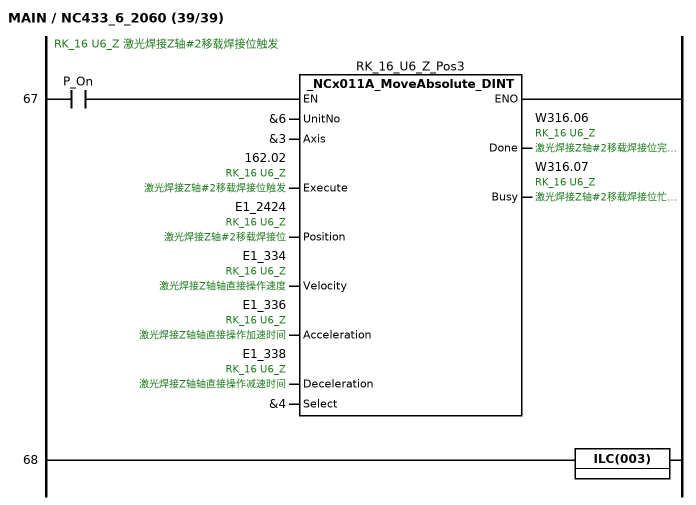
; [picture p264: MAIN / NC433_6_2060, rungs 67-68]
; rung 67: RK_16 U6_Z 激光焊接Z轴#2移载焊接位触发
LD P_On
CALL RK_16_U6_Z_Pos3 : _NCx011A_MoveAbsolute_DINT (UnitNo := &6, Axis := &3, Execute := 162.02, Position := E1_2424, Velocity := E1_334, Acceleration := E1_336, Deceleration := E1_338, Select := &4, Done => W316.06, Busy => W316.07)  ; RK_16 U6_Z 激光焊接Z轴#2移载焊接位触发, RK_16 U6_Z 激光焊接Z轴#2移载焊接位, RK_16 U6_Z 激光焊接Z轴轴直接操作速度, RK_16 U6_Z 激光焊接Z轴轴直接操作加速时间, RK_16 U6_Z 激光焊接Z轴轴直接操作减速时间, RK_16 U6_Z 激光焊接Z轴#2移载焊接位完成标志, RK_16 U6_Z 激光焊接Z轴#2移载焊接位忙标志
; rung 68
ILC(003)

### Section NC433_8_2080

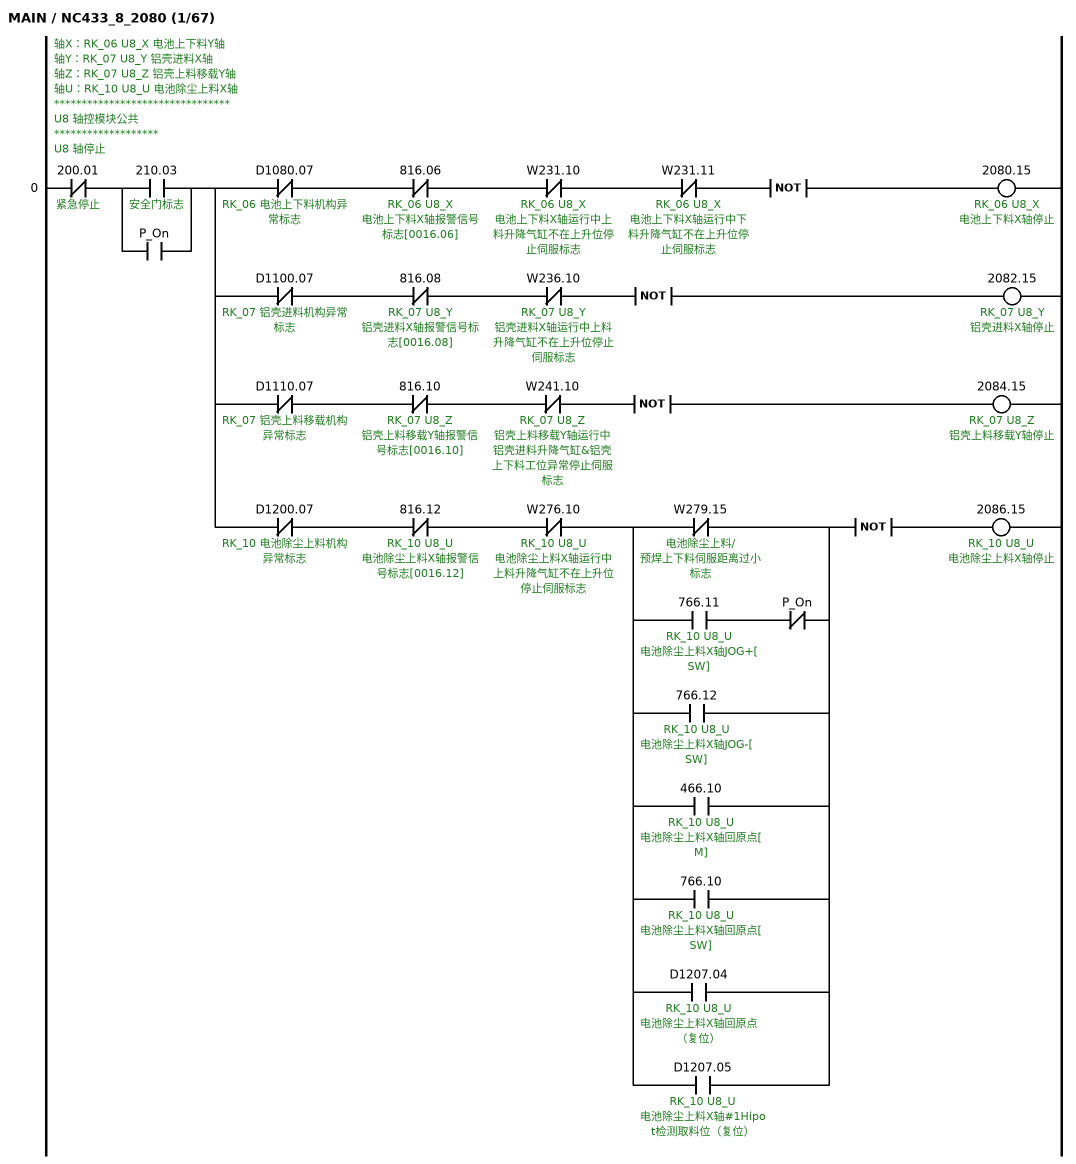
; rung 0: 轴X：RK_06 U8_X 电池上下料Y轴 / 轴Y：RK_07 U8_Y 铝壳进料X轴 / 轴Z：RK_07 U8_Z 铝壳上料移载Y轴 / 轴U：RK_10 U8_U 电池除尘上料X轴 / ******************************** / U8 轴控模块公共 / ******************* / U8 轴停止
LDNOT 200.01  ; 紧急停止
LD 210.03  ; 安全门标志
OR P_On
ANDLD
OUT TR0
ANDNOT D1080.07  ; RK_06 电池上下料机构异常标志
ANDNOT 816.06  ; RK_06 U8_X 电池上下料X轴报警信号标志[0016.06]
ANDNOT W231.10  ; RK_06 U8_X 电池上下料X轴运行中上料升降气缸不在上升位停止伺服标志
ANDNOT W231.11  ; RK_06 U8_X 电池上下料X轴运行中下料升降气缸不在上升位停止伺服标志
NOT(520)
OUT 2080.15  ; RK_06 U8_X 电池上下料X轴停止
LD TR0
ANDNOT D1100.07  ; RK_07 铝壳进料机构异常标志
ANDNOT 816.08  ; RK_07 U8_Y 铝壳进料X轴报警信号标志[0016.08]
ANDNOT W236.10  ; RK_07 U8_Y 铝壳进料X轴运行中上料升降气缸不在上升位停止伺服标志
NOT(520)
OUT 2082.15  ; RK_07 U8_Y 铝壳进料X轴停止
LD TR0
ANDNOT D1110.07  ; RK_07 铝壳上料移载机构异常标志
ANDNOT 816.10  ; RK_07 U8_Z 铝壳上料移载Y轴报警信号标志[0016.10]
ANDNOT W241.10  ; RK_07 U8_Z 铝壳上料移载Y轴运行中铝壳进料升降气缸&铝壳上下料工位异常停止伺服标志
NOT(520)
OUT 2084.15  ; RK_07 U8_Z 铝壳上料移载Y轴停止
LD TR0
ANDNOT D1200.07  ; RK_10 电池除尘上料机构异常标志
ANDNOT 816.12  ; RK_10 U8_U 电池除尘上料X轴报警信号标志[0016.12]
ANDNOT W276.10  ; RK_10 U8_U 电池除尘上料X轴运行中上料升降气缸不在上升位停止伺服标志
LDNOT W279.15  ; 电池除尘上料/预焊上下料伺服距离过小标志
LD 766.11  ; RK_10 U8_U 电池除尘上料X轴JOG+[SW]
ANDNOT P_On
ORLD
OR 766.12  ; RK_10 U8_U 电池除尘上料X轴JOG-[SW]
OR 466.10  ; RK_10 U8_U 电池除尘上料X轴回原点[M]
OR 766.10  ; RK_10 U8_U 电池除尘上料X轴回原点[SW]
OR D1207.04  ; RK_10 U8_U 电池除尘上料X轴回原点（复位）
OR D1207.05  ; RK_10 U8_U 电池除尘上料X轴#1Hipot检测取料位（复位）
ANDLD
NOT(520)
OUT 2086.15  ; RK_10 U8_U 电池除尘上料X轴停止

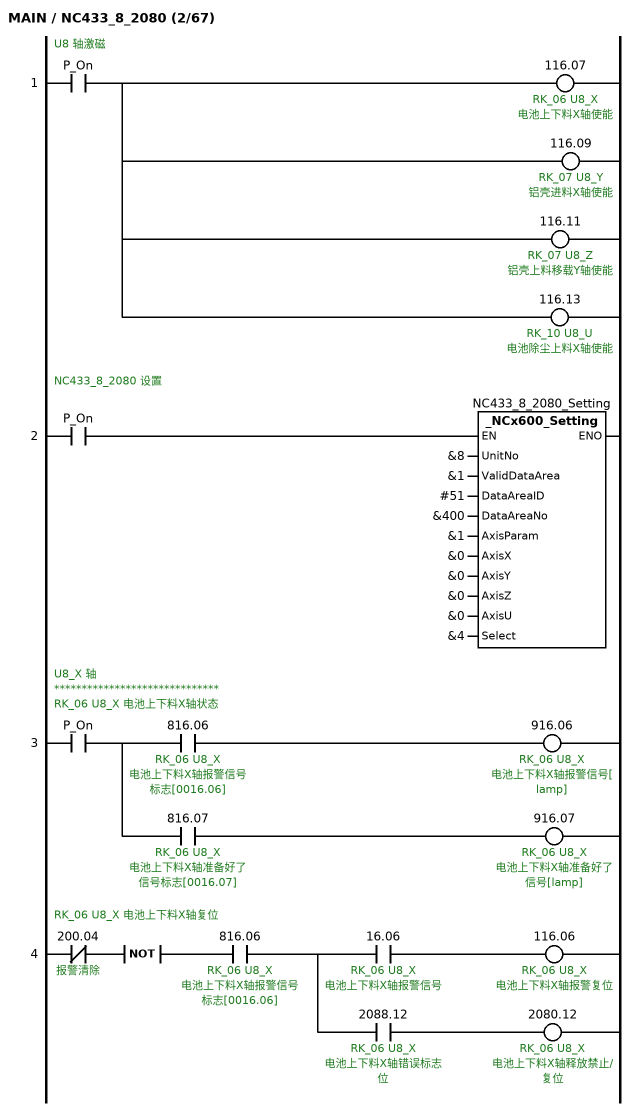
; rung 1: U8 轴激磁
LD P_On
OUT 116.07  ; RK_06 U8_X 电池上下料X轴使能
OUT 116.09  ; RK_07 U8_Y 铝壳进料X轴使能
OUT 116.11  ; RK_07 U8_Z 铝壳上料移载Y轴使能
OUT 116.13  ; RK_10 U8_U 电池除尘上料X轴使能
; rung 2: NC433_8_2080 设置
LD P_On
CALL NC433_8_2080_Setting : _NCx600_Setting (UnitNo := &8, ValidDataArea := &1, DataAreaID := #51, DataAreaNo := &400, AxisParam := &1, AxisX := &0, AxisY := &0, AxisZ := &0, AxisU := &0, Select := &4)
; rung 3: U8_X 轴 / ****************************** / RK_06 U8_X 电池上下料X轴状态
LD P_On
OUT TR0
AND 816.06  ; RK_06 U8_X 电池上下料X轴报警信号标志[0016.06]
OUT 916.06  ; RK_06 U8_X 电池上下料X轴报警信号[lamp]
LD TR0
AND 816.07  ; RK_06 U8_X 电池上下料X轴准备好了信号标志[0016.07]
OUT 916.07  ; RK_06 U8_X 电池上下料X轴准备好了信号[lamp]
; rung 4: RK_06 U8_X 电池上下料X轴复位
LDNOT 200.04  ; 报警清除
NOT(520)
AND 816.06  ; RK_06 U8_X 电池上下料X轴报警信号标志[0016.06]
OUT TR0
AND 16.06  ; RK_06 U8_X 电池上下料X轴报警信号
OUT 116.06  ; RK_06 U8_X 电池上下料X轴报警复位
LD TR0
AND 2088.12  ; RK_06 U8_X 电池上下料X轴错误标志位
OUT 2080.12  ; RK_06 U8_X 电池上下料X轴释放禁止/复位

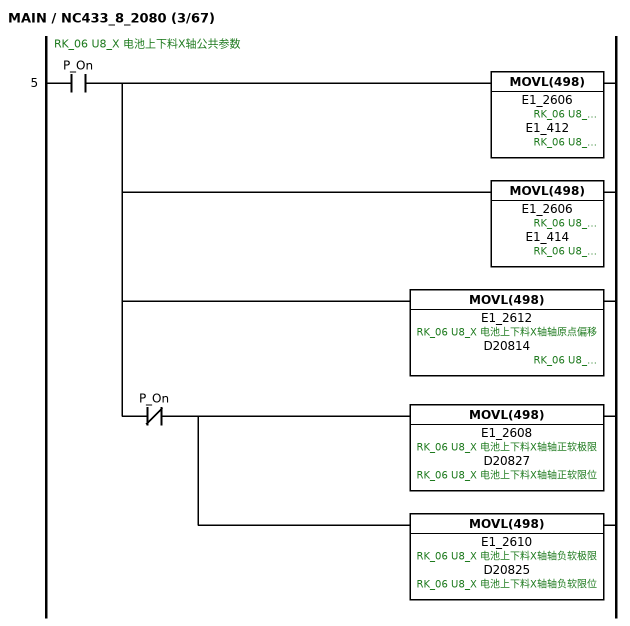
; rung 5: RK_06 U8_X 电池上下料X轴公共参数
LD P_On
MOVL(498) E1_2606 E1_412  ; RK_06 U8_X 电池上下料X轴轴加减速时间, RK_06 U8_X 电池上下料X轴轴直接操作加速时间
MOVL(498) E1_2606 E1_414  ; RK_06 U8_X 电池上下料X轴轴加减速时间, RK_06 U8_X 电池上下料X轴轴直接操作减速时间
MOVL(498) E1_2612 D20814  ; RK_06 U8_X 电池上下料X轴轴原点偏移, RK_06 U8_X 电池上下料X轴轴原点补偿值
ANDNOT P_On
MOVL(498) E1_2608 D20827  ; RK_06 U8_X 电池上下料X轴轴正软极限, RK_06 U8_X 电池上下料X轴轴正软限位
MOVL(498) E1_2610 D20825  ; RK_06 U8_X 电池上下料X轴轴负软极限, RK_06 U8_X 电池上下料X轴轴负软限位

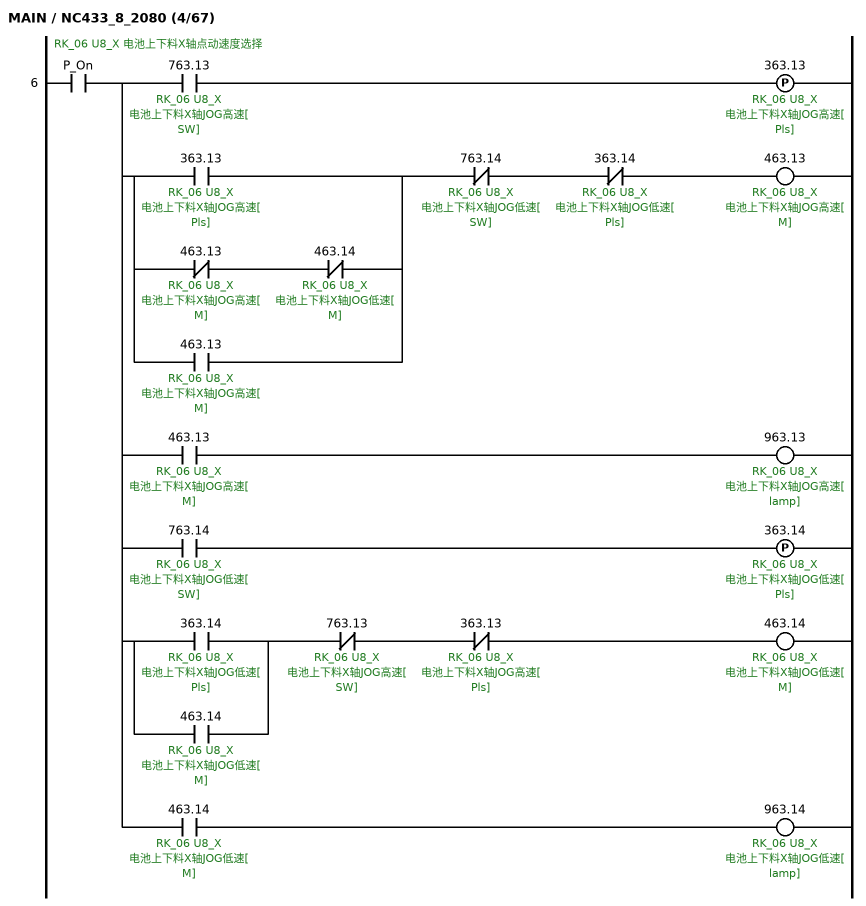
; rung 6: RK_06 U8_X 电池上下料X轴点动速度选择
LD P_On
OUT TR0
AND 763.13  ; RK_06 U8_X 电池上下料X轴JOG高速[SW]
DIFU(013) 363.13  ; RK_06 U8_X 电池上下料X轴JOG高速[Pls]
LD TR0
LD 363.13  ; RK_06 U8_X 电池上下料X轴JOG高速[Pls]
LDNOT 463.13  ; RK_06 U8_X 电池上下料X轴JOG高速[M]
ANDNOT 463.14  ; RK_06 U8_X 电池上下料X轴JOG低速[M]
ORLD
OR 463.13  ; RK_06 U8_X 电池上下料X轴JOG高速[M]
ANDLD
ANDNOT 763.14  ; RK_06 U8_X 电池上下料X轴JOG低速[SW]
ANDNOT 363.14  ; RK_06 U8_X 电池上下料X轴JOG低速[Pls]
OUT 463.13  ; RK_06 U8_X 电池上下料X轴JOG高速[M]
LD TR0
AND 463.13  ; RK_06 U8_X 电池上下料X轴JOG高速[M]
OUT 963.13  ; RK_06 U8_X 电池上下料X轴JOG高速[lamp]
LD TR0
AND 763.14  ; RK_06 U8_X 电池上下料X轴JOG低速[SW]
DIFU(013) 363.14  ; RK_06 U8_X 电池上下料X轴JOG低速[Pls]
LD TR0
LD 363.14  ; RK_06 U8_X 电池上下料X轴JOG低速[Pls]
OR 463.14  ; RK_06 U8_X 电池上下料X轴JOG低速[M]
ANDLD
ANDNOT 763.13  ; RK_06 U8_X 电池上下料X轴JOG高速[SW]
ANDNOT 363.13  ; RK_06 U8_X 电池上下料X轴JOG高速[Pls]
OUT 463.14  ; RK_06 U8_X 电池上下料X轴JOG低速[M]
LD TR0
AND 463.14  ; RK_06 U8_X 电池上下料X轴JOG低速[M]
OUT 963.14  ; RK_06 U8_X 电池上下料X轴JOG低速[lamp]

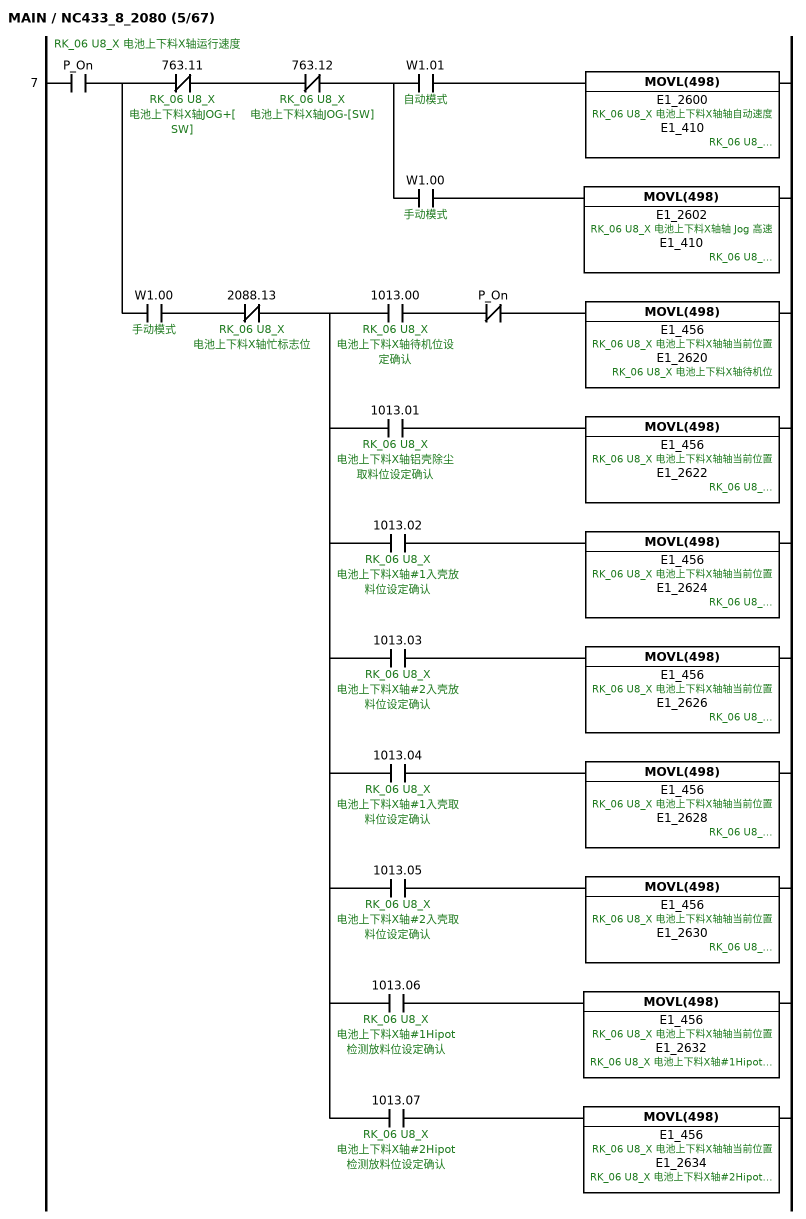
; rung 7: RK_06 U8_X 电池上下料X轴运行速度
LD P_On
OUT TR0
ANDNOT 763.11  ; RK_06 U8_X 电池上下料X轴JOG+[SW]
ANDNOT 763.12  ; RK_06 U8_X 电池上下料X轴JOG-[SW]
OUT TR1
AND W1.01  ; 自动模式
MOVL(498) E1_2600 E1_410  ; RK_06 U8_X 电池上下料X轴轴自动速度, RK_06 U8_X 电池上下料X轴轴直接操作速度
LD TR1
AND W1.00  ; 手动模式
MOVL(498) E1_2602 E1_410  ; RK_06 U8_X 电池上下料X轴轴 Jog 高速, RK_06 U8_X 电池上下料X轴轴直接操作速度
LD TR0
AND W1.00  ; 手动模式
ANDNOT 2088.13  ; RK_06 U8_X 电池上下料X轴忙标志位
OUT TR0
AND 1013.00  ; RK_06 U8_X 电池上下料X轴待机位设定确认
ANDNOT P_On
MOVL(498) E1_456 E1_2620  ; RK_06 U8_X 电池上下料X轴轴当前位置, RK_06 U8_X 电池上下料X轴待机位
LD TR0
AND 1013.01  ; RK_06 U8_X 电池上下料X轴铝壳除尘取料位设定确认
MOVL(498) E1_456 E1_2622  ; RK_06 U8_X 电池上下料X轴轴当前位置, RK_06 U8_X 电池上下料X轴铝壳除尘取料位
LD TR0
AND 1013.02  ; RK_06 U8_X 电池上下料X轴#1入壳放料位设定确认
MOVL(498) E1_456 E1_2624  ; RK_06 U8_X 电池上下料X轴轴当前位置, RK_06 U8_X 电池上下料X轴#1入壳放料位
LD TR0
AND 1013.03  ; RK_06 U8_X 电池上下料X轴#2入壳放料位设定确认
MOVL(498) E1_456 E1_2626  ; RK_06 U8_X 电池上下料X轴轴当前位置, RK_06 U8_X 电池上下料X轴#2入壳放料位
LD TR0
AND 1013.04  ; RK_06 U8_X 电池上下料X轴#1入壳取料位设定确认
MOVL(498) E1_456 E1_2628  ; RK_06 U8_X 电池上下料X轴轴当前位置, RK_06 U8_X 电池上下料X轴#1入壳取料位
LD TR0
AND 1013.05  ; RK_06 U8_X 电池上下料X轴#2入壳取料位设定确认
MOVL(498) E1_456 E1_2630  ; RK_06 U8_X 电池上下料X轴轴当前位置, RK_06 U8_X 电池上下料X轴#2入壳取料位
LD TR0
AND 1013.06  ; RK_06 U8_X 电池上下料X轴#1Hipot检测放料位设定确认
MOVL(498) E1_456 E1_2632  ; RK_06 U8_X 电池上下料X轴轴当前位置, RK_06 U8_X 电池上下料X轴#1Hipot检测放料位
LD TR0
AND 1013.07  ; RK_06 U8_X 电池上下料X轴#2Hipot检测放料位设定确认
MOVL(498) E1_456 E1_2634  ; RK_06 U8_X 电池上下料X轴轴当前位置, RK_06 U8_X 电池上下料X轴#2Hipot检测放料位

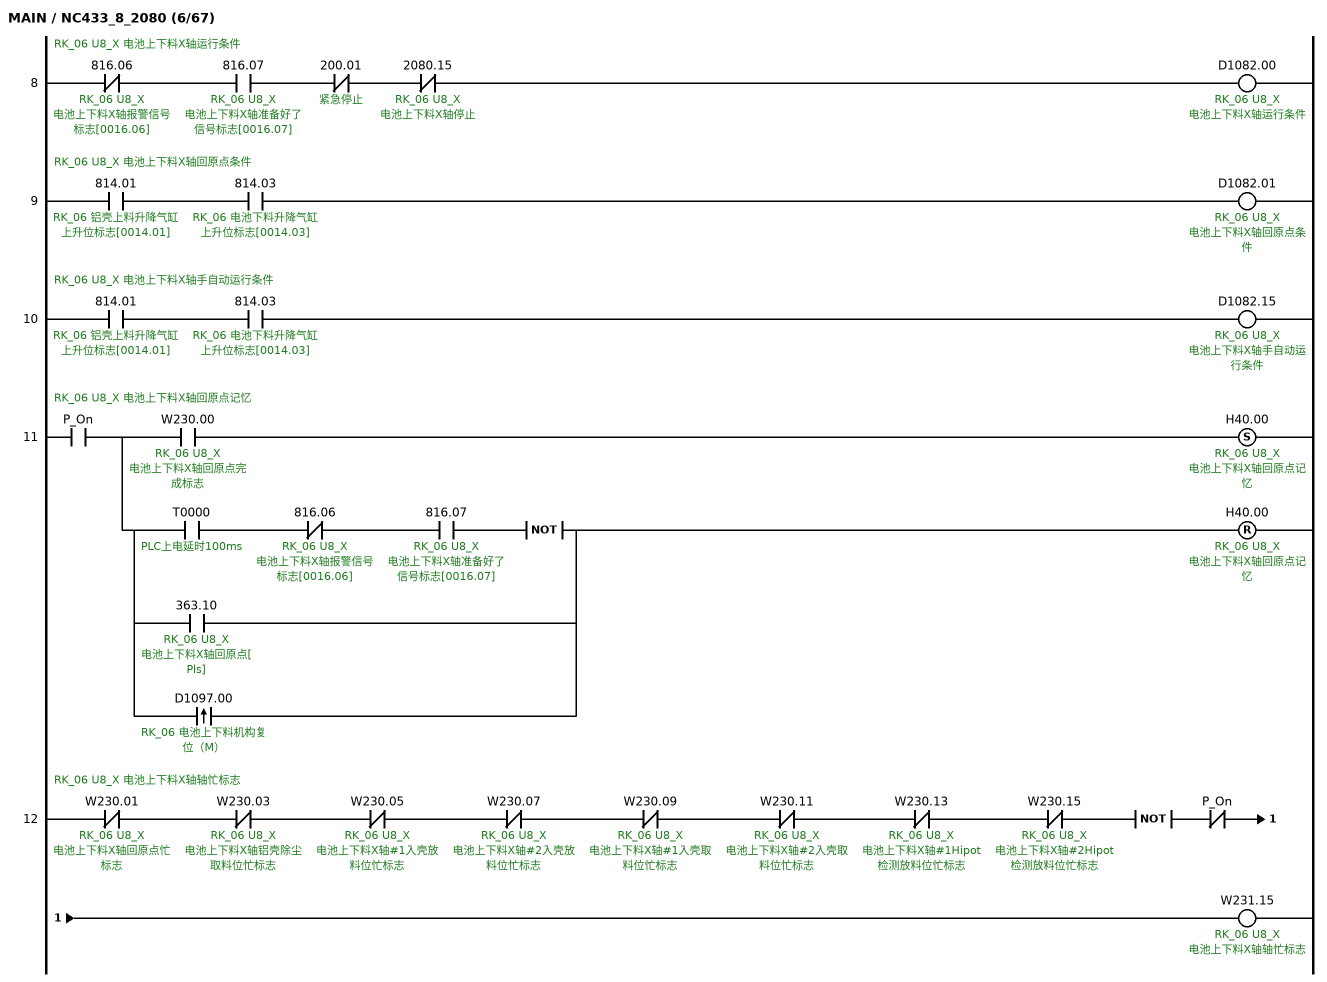
; rung 8: RK_06 U8_X 电池上下料X轴运行条件
LDNOT 816.06  ; RK_06 U8_X 电池上下料X轴报警信号标志[0016.06]
AND 816.07  ; RK_06 U8_X 电池上下料X轴准备好了信号标志[0016.07]
ANDNOT 200.01  ; 紧急停止
ANDNOT 2080.15  ; RK_06 U8_X 电池上下料X轴停止
OUT D1082.00  ; RK_06 U8_X 电池上下料X轴运行条件
; rung 9: RK_06 U8_X 电池上下料X轴回原点条件
LD 814.01  ; RK_06 铝壳上料升降气缸上升位标志[0014.01]
AND 814.03  ; RK_06 电池下料升降气缸上升位标志[0014.03]
OUT D1082.01  ; RK_06 U8_X 电池上下料X轴回原点条件
; rung 10: RK_06 U8_X 电池上下料X轴手自动运行条件
LD 814.01  ; RK_06 铝壳上料升降气缸上升位标志[0014.01]
AND 814.03  ; RK_06 电池下料升降气缸上升位标志[0014.03]
OUT D1082.15  ; RK_06 U8_X 电池上下料X轴手自动运行条件
; rung 11: RK_06 U8_X 电池上下料X轴回原点记忆
LD P_On
OUT TR0
AND W230.00  ; RK_06 U8_X 电池上下料X轴回原点完成标志
SET H40.00  ; RK_06 U8_X 电池上下料X轴回原点记忆
LD TR0
LD T0000  ; PLC上电延时100ms
ANDNOT 816.06  ; RK_06 U8_X 电池上下料X轴报警信号标志[0016.06]
AND 816.07  ; RK_06 U8_X 电池上下料X轴准备好了信号标志[0016.07]
NOT(520)
OR 363.10  ; RK_06 U8_X 电池上下料X轴回原点[Pls]
@OR D1097.00  ; RK_06 电池上下料机构复位（M）
ANDLD
RSET H40.00  ; RK_06 U8_X 电池上下料X轴回原点记忆
; rung 12: RK_06 U8_X 电池上下料X轴轴忙标志
LDNOT W230.01  ; RK_06 U8_X 电池上下料X轴回原点忙标志
ANDNOT W230.03  ; RK_06 U8_X 电池上下料X轴铝壳除尘取料位忙标志
ANDNOT W230.05  ; RK_06 U8_X 电池上下料X轴#1入壳放料位忙标志
ANDNOT W230.07  ; RK_06 U8_X 电池上下料X轴#2入壳放料位忙标志
ANDNOT W230.09  ; RK_06 U8_X 电池上下料X轴#1入壳取料位忙标志
ANDNOT W230.11  ; RK_06 U8_X 电池上下料X轴#2入壳取料位忙标志
ANDNOT W230.13  ; RK_06 U8_X 电池上下料X轴#1Hipot检测放料位忙标志
ANDNOT W230.15  ; RK_06 U8_X 电池上下料X轴#2Hipot检测放料位忙标志
NOT(520)
ANDNOT P_On
OUT W231.15  ; RK_06 U8_X 电池上下料X轴轴忙标志

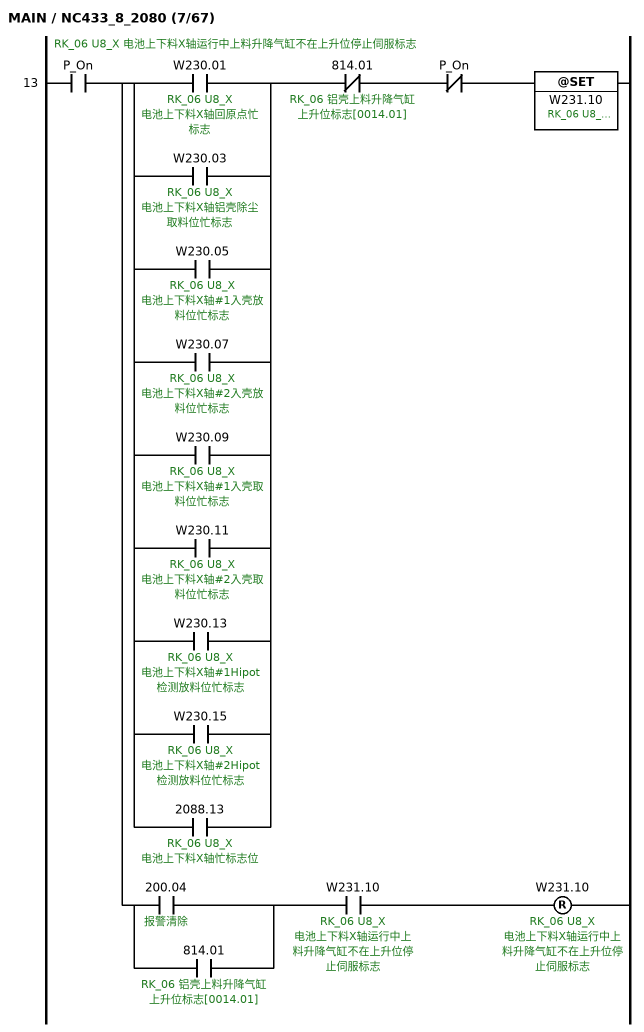
; rung 13: RK_06 U8_X 电池上下料X轴运行中上料升降气缸不在上升位停止伺服标志
LD P_On
OUT TR0
LD W230.01  ; RK_06 U8_X 电池上下料X轴回原点忙标志
OR W230.03  ; RK_06 U8_X 电池上下料X轴铝壳除尘取料位忙标志
OR W230.05  ; RK_06 U8_X 电池上下料X轴#1入壳放料位忙标志
OR W230.07  ; RK_06 U8_X 电池上下料X轴#2入壳放料位忙标志
OR W230.09  ; RK_06 U8_X 电池上下料X轴#1入壳取料位忙标志
OR W230.11  ; RK_06 U8_X 电池上下料X轴#2入壳取料位忙标志
OR W230.13  ; RK_06 U8_X 电池上下料X轴#1Hipot检测放料位忙标志
OR W230.15  ; RK_06 U8_X 电池上下料X轴#2Hipot检测放料位忙标志
OR 2088.13  ; RK_06 U8_X 电池上下料X轴忙标志位
ANDLD
ANDNOT 814.01  ; RK_06 铝壳上料升降气缸上升位标志[0014.01]
ANDNOT P_On
@SET W231.10  ; RK_06 U8_X 电池上下料X轴运行中上料升降气缸不在上升位停止伺服标志  // 增加相应报警信息
LD TR0
LD 200.04  ; 报警清除
OR 814.01  ; RK_06 铝壳上料升降气缸上升位标志[0014.01]
ANDLD
AND W231.10  ; RK_06 U8_X 电池上下料X轴运行中上料升降气缸不在上升位停止伺服标志
RSET W231.10  ; RK_06 U8_X 电池上下料X轴运行中上料升降气缸不在上升位停止伺服标志

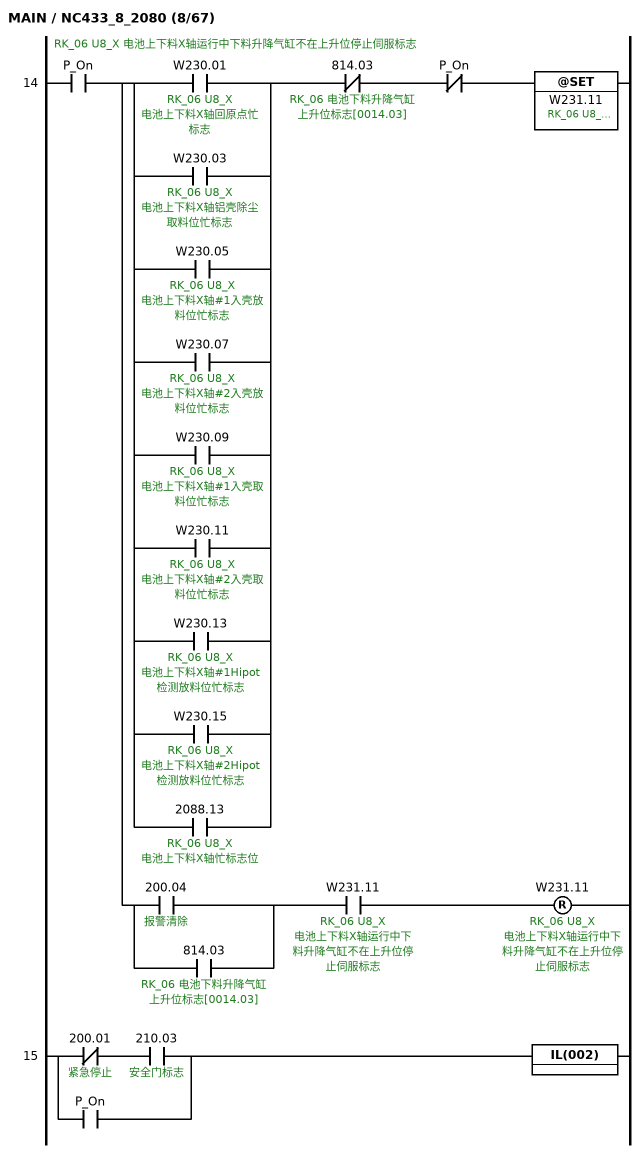
; rung 14: RK_06 U8_X 电池上下料X轴运行中下料升降气缸不在上升位停止伺服标志
LD P_On
OUT TR0
LD W230.01  ; RK_06 U8_X 电池上下料X轴回原点忙标志
OR W230.03  ; RK_06 U8_X 电池上下料X轴铝壳除尘取料位忙标志
OR W230.05  ; RK_06 U8_X 电池上下料X轴#1入壳放料位忙标志
OR W230.07  ; RK_06 U8_X 电池上下料X轴#2入壳放料位忙标志
OR W230.09  ; RK_06 U8_X 电池上下料X轴#1入壳取料位忙标志
OR W230.11  ; RK_06 U8_X 电池上下料X轴#2入壳取料位忙标志
OR W230.13  ; RK_06 U8_X 电池上下料X轴#1Hipot检测放料位忙标志
OR W230.15  ; RK_06 U8_X 电池上下料X轴#2Hipot检测放料位忙标志
OR 2088.13  ; RK_06 U8_X 电池上下料X轴忙标志位
ANDLD
ANDNOT 814.03  ; RK_06 电池下料升降气缸上升位标志[0014.03]
ANDNOT P_On
@SET W231.11  ; RK_06 U8_X 电池上下料X轴运行中下料升降气缸不在上升位停止伺服标志  // 增加相应报警信息
LD TR0
LD 200.04  ; 报警清除
OR 814.03  ; RK_06 电池下料升降气缸上升位标志[0014.03]
ANDLD
AND W231.11  ; RK_06 U8_X 电池上下料X轴运行中下料升降气缸不在上升位停止伺服标志
RSET W231.11  ; RK_06 U8_X 电池上下料X轴运行中下料升降气缸不在上升位停止伺服标志
; rung 15
LDNOT 200.01  ; 紧急停止
AND 210.03  ; 安全门标志
OR P_On
IL(002)

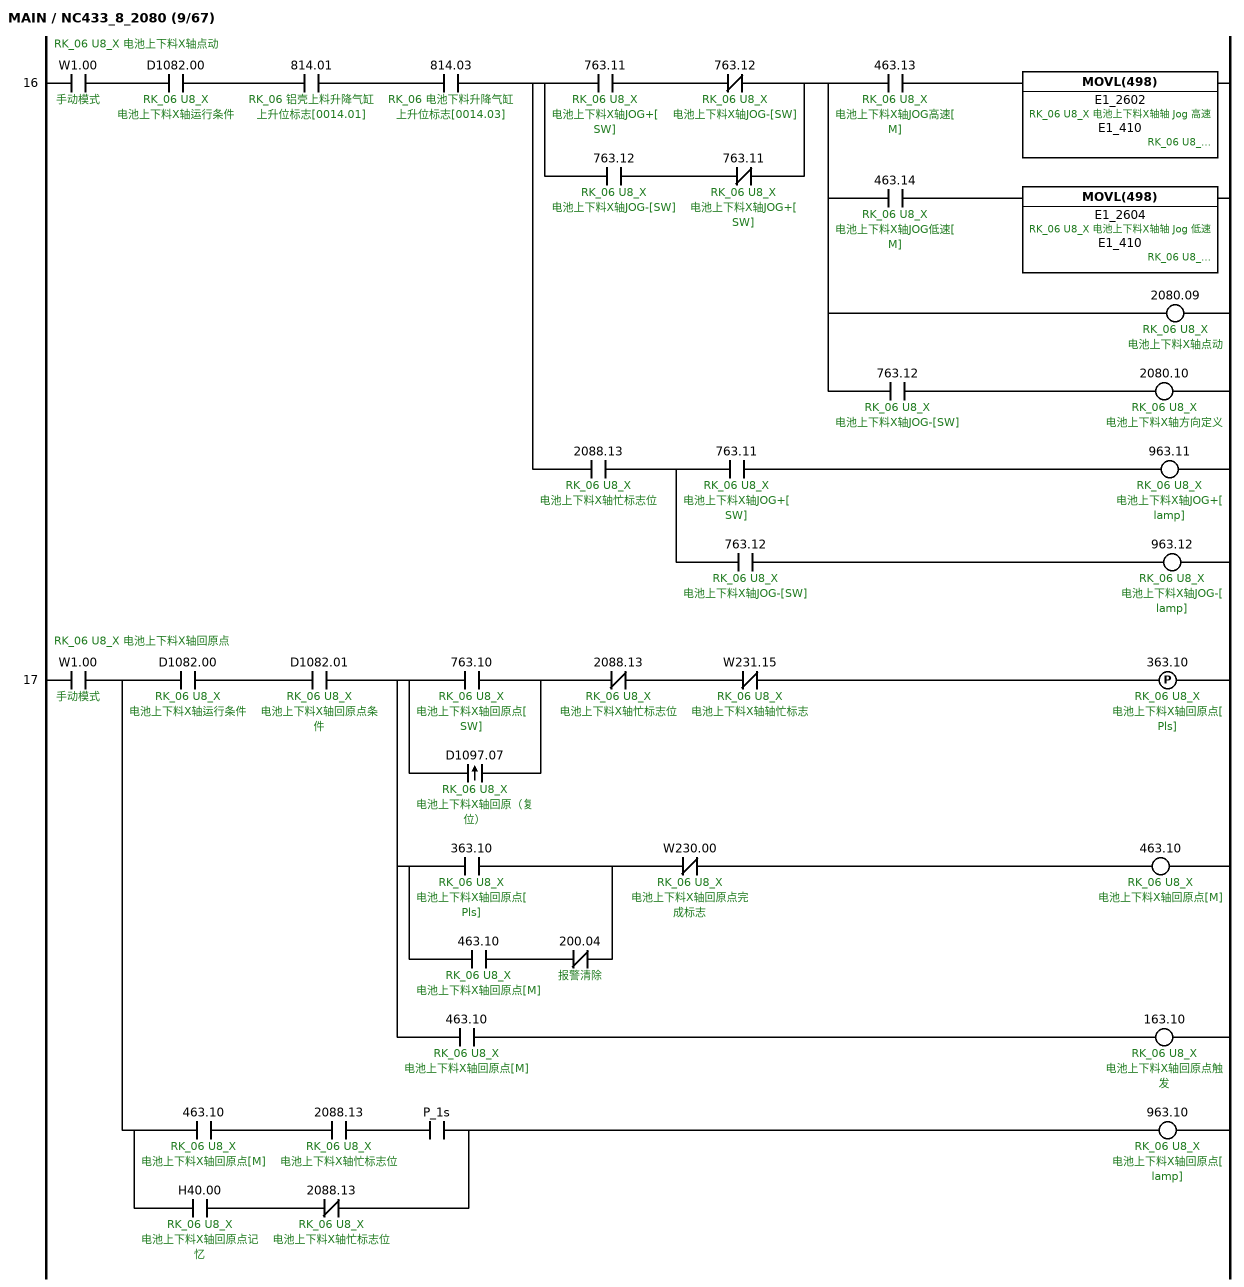
; rung 16: RK_06 U8_X 电池上下料X轴点动
LD W1.00  ; 手动模式
AND D1082.00  ; RK_06 U8_X 电池上下料X轴运行条件
AND 814.01  ; RK_06 铝壳上料升降气缸上升位标志[0014.01]
AND 814.03  ; RK_06 电池下料升降气缸上升位标志[0014.03]
OUT TR0
LD 763.11  ; RK_06 U8_X 电池上下料X轴JOG+[SW]
ANDNOT 763.12  ; RK_06 U8_X 电池上下料X轴JOG-[SW]
LD 763.12  ; RK_06 U8_X 电池上下料X轴JOG-[SW]
ANDNOT 763.11  ; RK_06 U8_X 电池上下料X轴JOG+[SW]
ORLD
ANDLD
OUT TR1
AND 463.13  ; RK_06 U8_X 电池上下料X轴JOG高速[M]
MOVL(498) E1_2602 E1_410  ; RK_06 U8_X 电池上下料X轴轴 Jog 高速, RK_06 U8_X 电池上下料X轴轴直接操作速度
LD TR1
AND 463.14  ; RK_06 U8_X 电池上下料X轴JOG低速[M]
MOVL(498) E1_2604 E1_410  ; RK_06 U8_X 电池上下料X轴轴 Jog 低速, RK_06 U8_X 电池上下料X轴轴直接操作速度
LD TR1
OUT 2080.09  ; RK_06 U8_X 电池上下料X轴点动
AND 763.12  ; RK_06 U8_X 电池上下料X轴JOG-[SW]
OUT 2080.10  ; RK_06 U8_X 电池上下料X轴方向定义
LD TR0
AND 2088.13  ; RK_06 U8_X 电池上下料X轴忙标志位
OUT TR0
AND 763.11  ; RK_06 U8_X 电池上下料X轴JOG+[SW]
OUT 963.11  ; RK_06 U8_X 电池上下料X轴JOG+[lamp]
LD TR0
AND 763.12  ; RK_06 U8_X 电池上下料X轴JOG-[SW]
OUT 963.12  ; RK_06 U8_X 电池上下料X轴JOG-[lamp]
; rung 17: RK_06 U8_X 电池上下料X轴回原点
LD W1.00  ; 手动模式
OUT TR0
AND D1082.00  ; RK_06 U8_X 电池上下料X轴运行条件
AND D1082.01  ; RK_06 U8_X 电池上下料X轴回原点条件
OUT TR1
LD 763.10  ; RK_06 U8_X 电池上下料X轴回原点[SW]
@OR D1097.07  ; RK_06 U8_X 电池上下料X轴回原（复位）
ANDLD
ANDNOT 2088.13  ; RK_06 U8_X 电池上下料X轴忙标志位
ANDNOT W231.15  ; RK_06 U8_X 电池上下料X轴轴忙标志
DIFU(013) 363.10  ; RK_06 U8_X 电池上下料X轴回原点[Pls]
LD TR1
LD 363.10  ; RK_06 U8_X 电池上下料X轴回原点[Pls]
LD 463.10  ; RK_06 U8_X 电池上下料X轴回原点[M]
ANDNOT 200.04  ; 报警清除
ORLD
ANDLD
ANDNOT W230.00  ; RK_06 U8_X 电池上下料X轴回原点完成标志
OUT 463.10  ; RK_06 U8_X 电池上下料X轴回原点[M]
LD TR1
AND 463.10  ; RK_06 U8_X 电池上下料X轴回原点[M]
OUT 163.10  ; RK_06 U8_X 电池上下料X轴回原点触发
LD TR0
LD 463.10  ; RK_06 U8_X 电池上下料X轴回原点[M]
AND 2088.13  ; RK_06 U8_X 电池上下料X轴忙标志位
AND P_1s
LD H40.00  ; RK_06 U8_X 电池上下料X轴回原点记忆
ANDNOT 2088.13  ; RK_06 U8_X 电池上下料X轴忙标志位
ORLD
ANDLD
OUT 963.10  ; RK_06 U8_X 电池上下料X轴回原点[lamp]

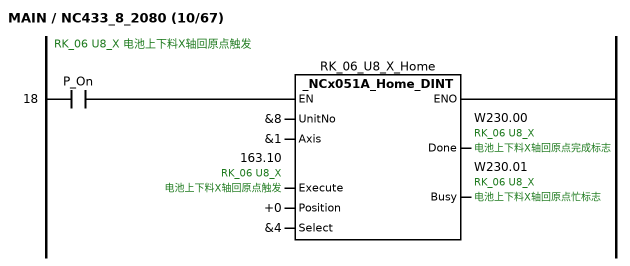
; rung 18: RK_06 U8_X 电池上下料X轴回原点触发
LD P_On
CALL RK_06_U8_X_Home : _NCx051A_Home_DINT (UnitNo := &8, Axis := &1, Execute := 163.10, Position := +0, Select := &4, Done => W230.00, Busy => W230.01)  ; RK_06 U8_X 电池上下料X轴回原点触发, RK_06 U8_X 电池上下料X轴回原点完成标志, RK_06 U8_X 电池上下料X轴回原点忙标志

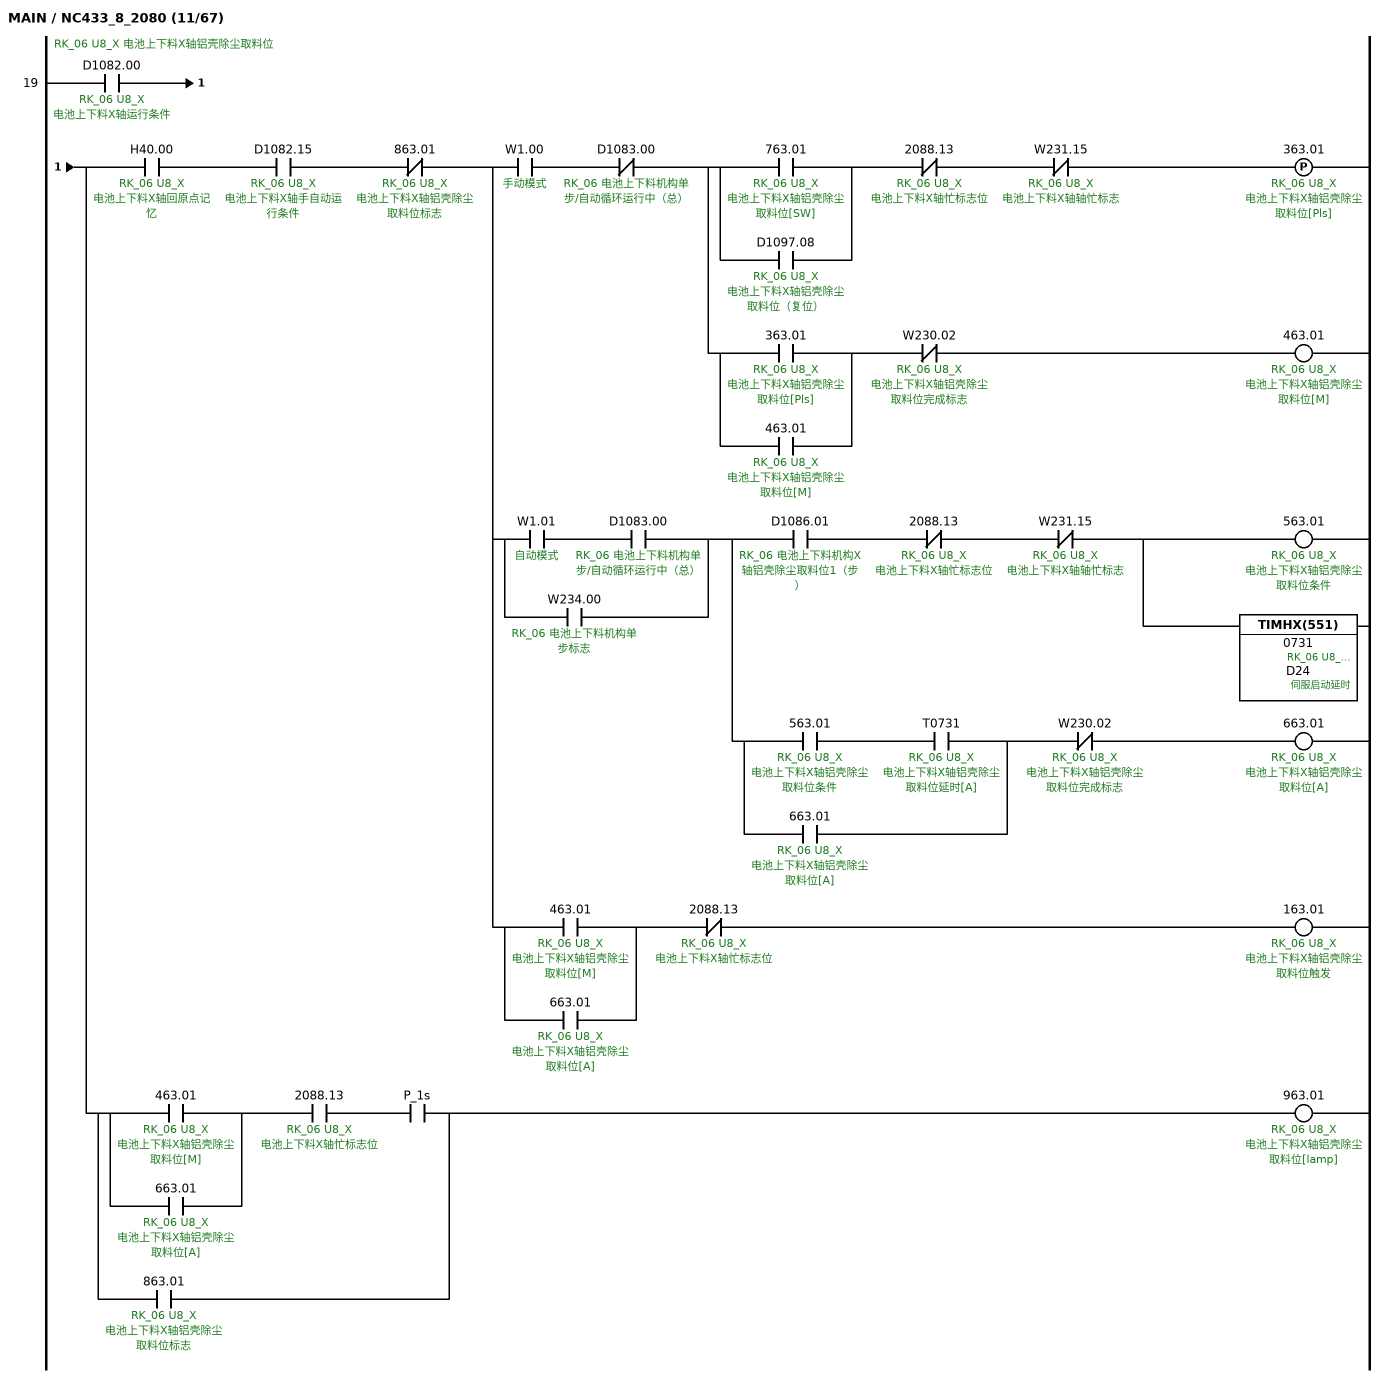
; rung 19: RK_06 U8_X 电池上下料X轴铝壳除尘取料位
LD D1082.00  ; RK_06 U8_X 电池上下料X轴运行条件
OUT TR0
AND H40.00  ; RK_06 U8_X 电池上下料X轴回原点记忆
AND D1082.15  ; RK_06 U8_X 电池上下料X轴手自动运行条件
ANDNOT 863.01  ; RK_06 U8_X 电池上下料X轴铝壳除尘取料位标志
OUT TR1
AND W1.00  ; 手动模式
ANDNOT D1083.00  ; RK_06 电池上下料机构单步/自动循环运行中（总）
OUT TR2
LD 763.01  ; RK_06 U8_X 电池上下料X轴铝壳除尘取料位[SW]
OR D1097.08  ; RK_06 U8_X 电池上下料X轴铝壳除尘取料位（复位）
ANDLD
ANDNOT 2088.13  ; RK_06 U8_X 电池上下料X轴忙标志位
ANDNOT W231.15  ; RK_06 U8_X 电池上下料X轴轴忙标志
DIFU(013) 363.01  ; RK_06 U8_X 电池上下料X轴铝壳除尘取料位[Pls]
LD TR2
LD 363.01  ; RK_06 U8_X 电池上下料X轴铝壳除尘取料位[Pls]
OR 463.01  ; RK_06 U8_X 电池上下料X轴铝壳除尘取料位[M]
ANDLD
ANDNOT W230.02  ; RK_06 U8_X 电池上下料X轴铝壳除尘取料位完成标志
OUT 463.01  ; RK_06 U8_X 电池上下料X轴铝壳除尘取料位[M]
LD TR1
LD W1.01  ; 自动模式
AND D1083.00  ; RK_06 电池上下料机构单步/自动循环运行中（总）
OR W234.00  ; RK_06 电池上下料机构单步标志
ANDLD
OUT TR2
AND D1086.01  ; RK_06 电池上下料机构X轴铝壳除尘取料位1（步）
ANDNOT 2088.13  ; RK_06 U8_X 电池上下料X轴忙标志位
ANDNOT W231.15  ; RK_06 U8_X 电池上下料X轴轴忙标志
OUT 563.01  ; RK_06 U8_X 电池上下料X轴铝壳除尘取料位条件
TIMHX(551) 0731 D24  ; 伺服启动延时, RK_06 U8_X 电池上下料X轴铝壳除尘取料位延时[A]
LD TR2
LD 563.01  ; RK_06 U8_X 电池上下料X轴铝壳除尘取料位条件
AND T0731  ; RK_06 U8_X 电池上下料X轴铝壳除尘取料位延时[A]
OR 663.01  ; RK_06 U8_X 电池上下料X轴铝壳除尘取料位[A]
ANDLD
ANDNOT W230.02  ; RK_06 U8_X 电池上下料X轴铝壳除尘取料位完成标志
OUT 663.01  ; RK_06 U8_X 电池上下料X轴铝壳除尘取料位[A]
LD TR1
LD 463.01  ; RK_06 U8_X 电池上下料X轴铝壳除尘取料位[M]
OR 663.01  ; RK_06 U8_X 电池上下料X轴铝壳除尘取料位[A]
ANDLD
ANDNOT 2088.13  ; RK_06 U8_X 电池上下料X轴忙标志位
OUT 163.01  ; RK_06 U8_X 电池上下料X轴铝壳除尘取料位触发
LD TR0
LD 463.01  ; RK_06 U8_X 电池上下料X轴铝壳除尘取料位[M]
OR 663.01  ; RK_06 U8_X 电池上下料X轴铝壳除尘取料位[A]
AND 2088.13  ; RK_06 U8_X 电池上下料X轴忙标志位
AND P_1s
OR 863.01  ; RK_06 U8_X 电池上下料X轴铝壳除尘取料位标志
ANDLD
OUT 963.01  ; RK_06 U8_X 电池上下料X轴铝壳除尘取料位[lamp]

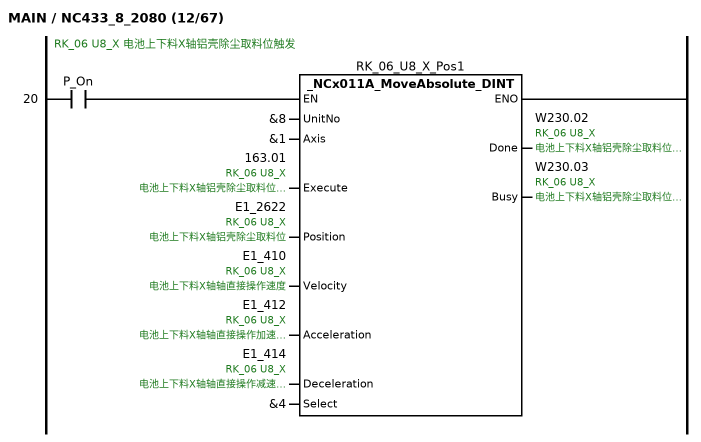
; rung 20: RK_06 U8_X 电池上下料X轴铝壳除尘取料位触发
LD P_On
CALL RK_06_U8_X_Pos1 : _NCx011A_MoveAbsolute_DINT (UnitNo := &8, Axis := &1, Execute := 163.01, Position := E1_2622, Velocity := E1_410, Acceleration := E1_412, Deceleration := E1_414, Select := &4, Done => W230.02, Busy => W230.03)  ; RK_06 U8_X 电池上下料X轴铝壳除尘取料位触发, RK_06 U8_X 电池上下料X轴铝壳除尘取料位, RK_06 U8_X 电池上下料X轴轴直接操作速度, RK_06 U8_X 电池上下料X轴轴直接操作加速时间, RK_06 U8_X 电池上下料X轴轴直接操作减速时间, RK_06 U8_X 电池上下料X轴铝壳除尘取料位完成标志, RK_06 U8_X 电池上下料X轴铝壳除尘取料位忙标志

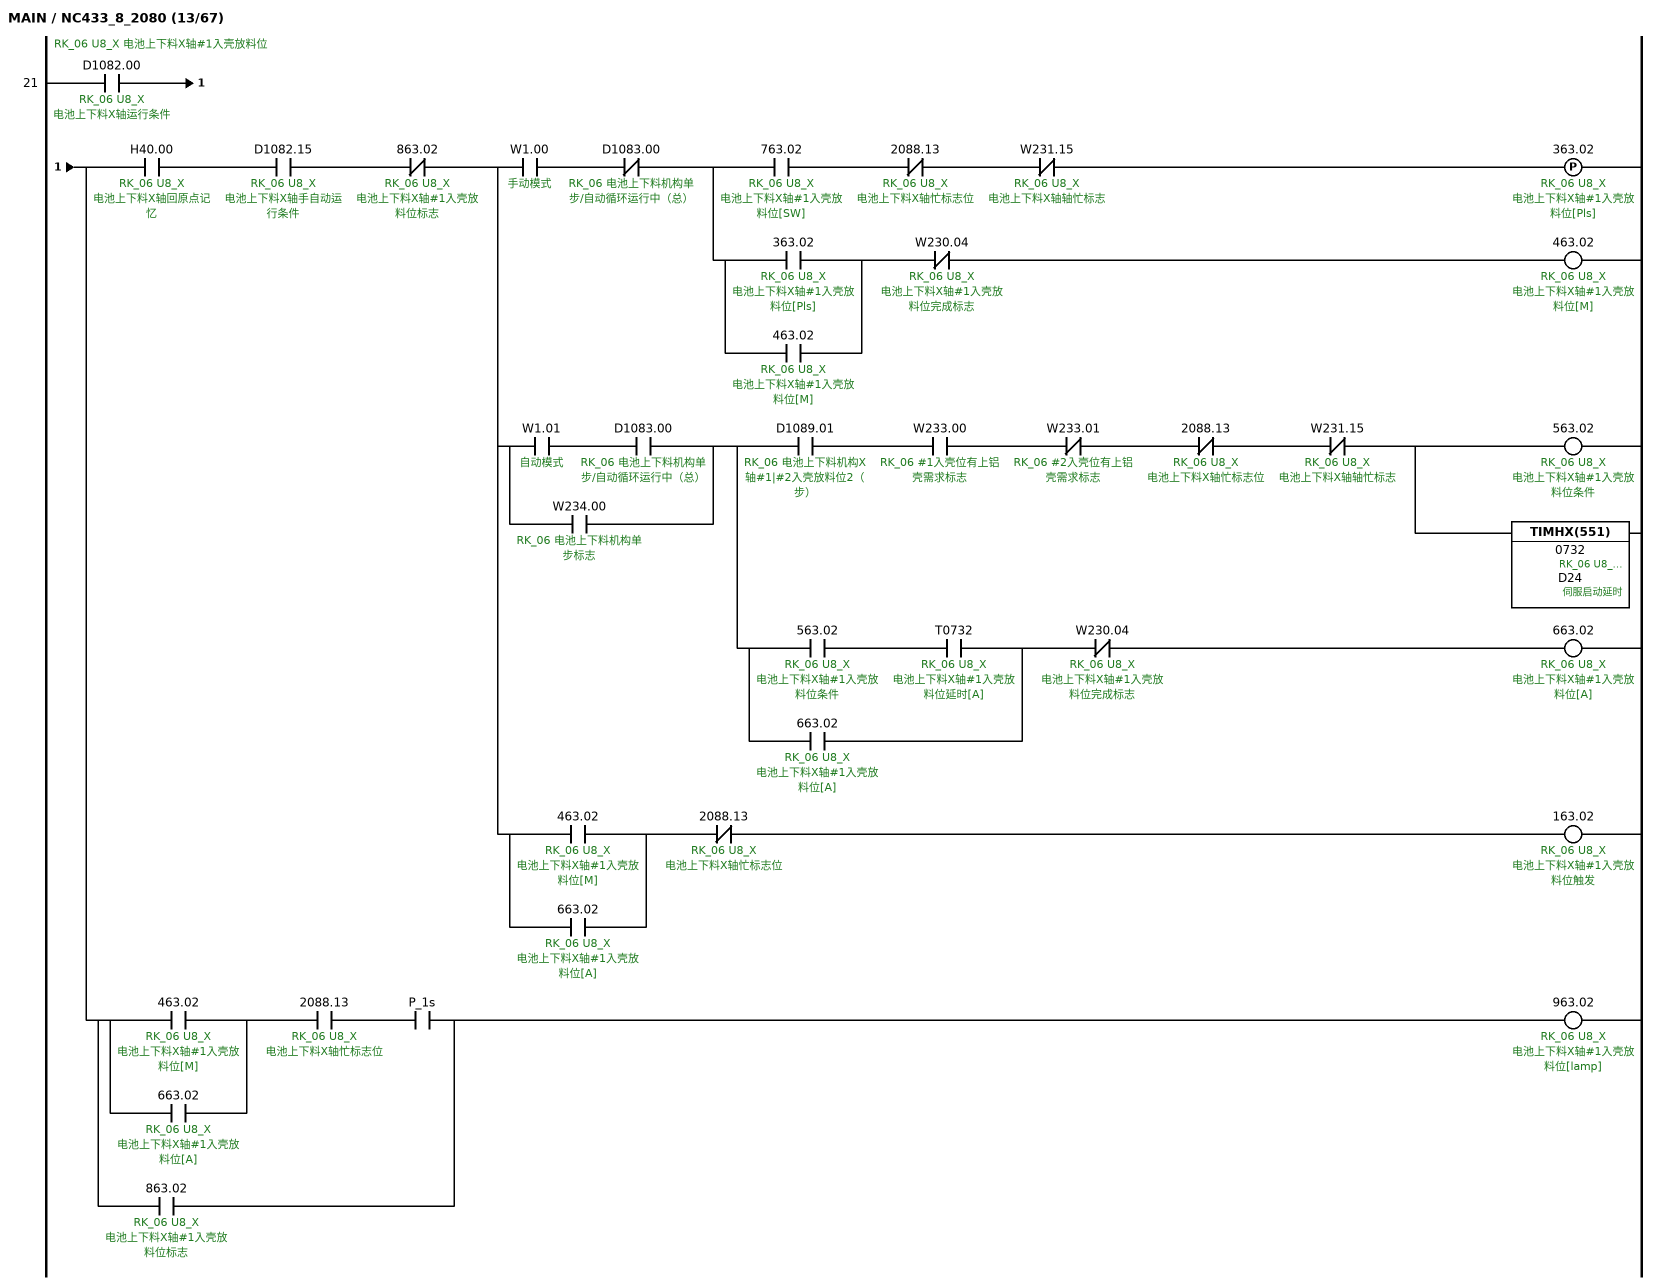
; rung 21: RK_06 U8_X 电池上下料X轴#1入壳放料位
LD D1082.00  ; RK_06 U8_X 电池上下料X轴运行条件
OUT TR0
AND H40.00  ; RK_06 U8_X 电池上下料X轴回原点记忆
AND D1082.15  ; RK_06 U8_X 电池上下料X轴手自动运行条件
ANDNOT 863.02  ; RK_06 U8_X 电池上下料X轴#1入壳放料位标志
OUT TR1
AND W1.00  ; 手动模式
ANDNOT D1083.00  ; RK_06 电池上下料机构单步/自动循环运行中（总）
OUT TR2
AND 763.02  ; RK_06 U8_X 电池上下料X轴#1入壳放料位[SW]
ANDNOT 2088.13  ; RK_06 U8_X 电池上下料X轴忙标志位
ANDNOT W231.15  ; RK_06 U8_X 电池上下料X轴轴忙标志
DIFU(013) 363.02  ; RK_06 U8_X 电池上下料X轴#1入壳放料位[Pls]
LD TR2
LD 363.02  ; RK_06 U8_X 电池上下料X轴#1入壳放料位[Pls]
OR 463.02  ; RK_06 U8_X 电池上下料X轴#1入壳放料位[M]
ANDLD
ANDNOT W230.04  ; RK_06 U8_X 电池上下料X轴#1入壳放料位完成标志
OUT 463.02  ; RK_06 U8_X 电池上下料X轴#1入壳放料位[M]
LD TR1
LD W1.01  ; 自动模式
AND D1083.00  ; RK_06 电池上下料机构单步/自动循环运行中（总）
OR W234.00  ; RK_06 电池上下料机构单步标志
ANDLD
OUT TR2
AND D1089.01  ; RK_06 电池上下料机构X轴#1|#2入壳放料位2（步）
AND W233.00  ; RK_06 #1入壳位有上铝壳需求标志
ANDNOT W233.01  ; RK_06 #2入壳位有上铝壳需求标志
ANDNOT 2088.13  ; RK_06 U8_X 电池上下料X轴忙标志位
ANDNOT W231.15  ; RK_06 U8_X 电池上下料X轴轴忙标志
OUT 563.02  ; RK_06 U8_X 电池上下料X轴#1入壳放料位条件
TIMHX(551) 0732 D24  ; 伺服启动延时, RK_06 U8_X 电池上下料X轴#1入壳放料位延时[A]
LD TR2
LD 563.02  ; RK_06 U8_X 电池上下料X轴#1入壳放料位条件
AND T0732  ; RK_06 U8_X 电池上下料X轴#1入壳放料位延时[A]
OR 663.02  ; RK_06 U8_X 电池上下料X轴#1入壳放料位[A]
ANDLD
ANDNOT W230.04  ; RK_06 U8_X 电池上下料X轴#1入壳放料位完成标志
OUT 663.02  ; RK_06 U8_X 电池上下料X轴#1入壳放料位[A]
LD TR1
LD 463.02  ; RK_06 U8_X 电池上下料X轴#1入壳放料位[M]
OR 663.02  ; RK_06 U8_X 电池上下料X轴#1入壳放料位[A]
ANDLD
ANDNOT 2088.13  ; RK_06 U8_X 电池上下料X轴忙标志位
OUT 163.02  ; RK_06 U8_X 电池上下料X轴#1入壳放料位触发
LD TR0
LD 463.02  ; RK_06 U8_X 电池上下料X轴#1入壳放料位[M]
OR 663.02  ; RK_06 U8_X 电池上下料X轴#1入壳放料位[A]
AND 2088.13  ; RK_06 U8_X 电池上下料X轴忙标志位
AND P_1s
OR 863.02  ; RK_06 U8_X 电池上下料X轴#1入壳放料位标志
ANDLD
OUT 963.02  ; RK_06 U8_X 电池上下料X轴#1入壳放料位[lamp]

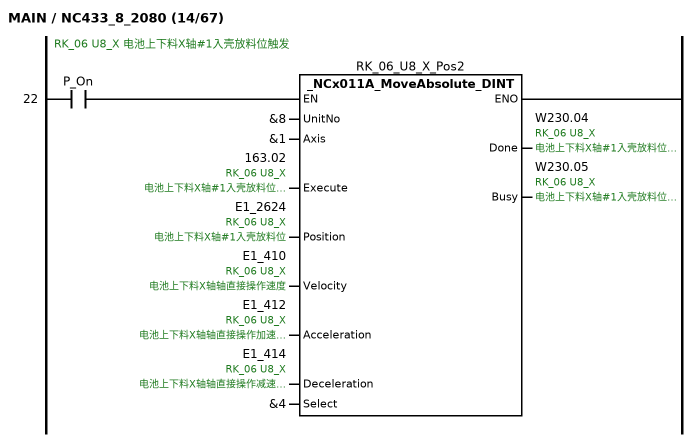
; rung 22: RK_06 U8_X 电池上下料X轴#1入壳放料位触发
LD P_On
CALL RK_06_U8_X_Pos2 : _NCx011A_MoveAbsolute_DINT (UnitNo := &8, Axis := &1, Execute := 163.02, Position := E1_2624, Velocity := E1_410, Acceleration := E1_412, Deceleration := E1_414, Select := &4, Done => W230.04, Busy => W230.05)  ; RK_06 U8_X 电池上下料X轴#1入壳放料位触发, RK_06 U8_X 电池上下料X轴#1入壳放料位, RK_06 U8_X 电池上下料X轴轴直接操作速度, RK_06 U8_X 电池上下料X轴轴直接操作加速时间, RK_06 U8_X 电池上下料X轴轴直接操作减速时间, RK_06 U8_X 电池上下料X轴#1入壳放料位完成标志, RK_06 U8_X 电池上下料X轴#1入壳放料位忙标志

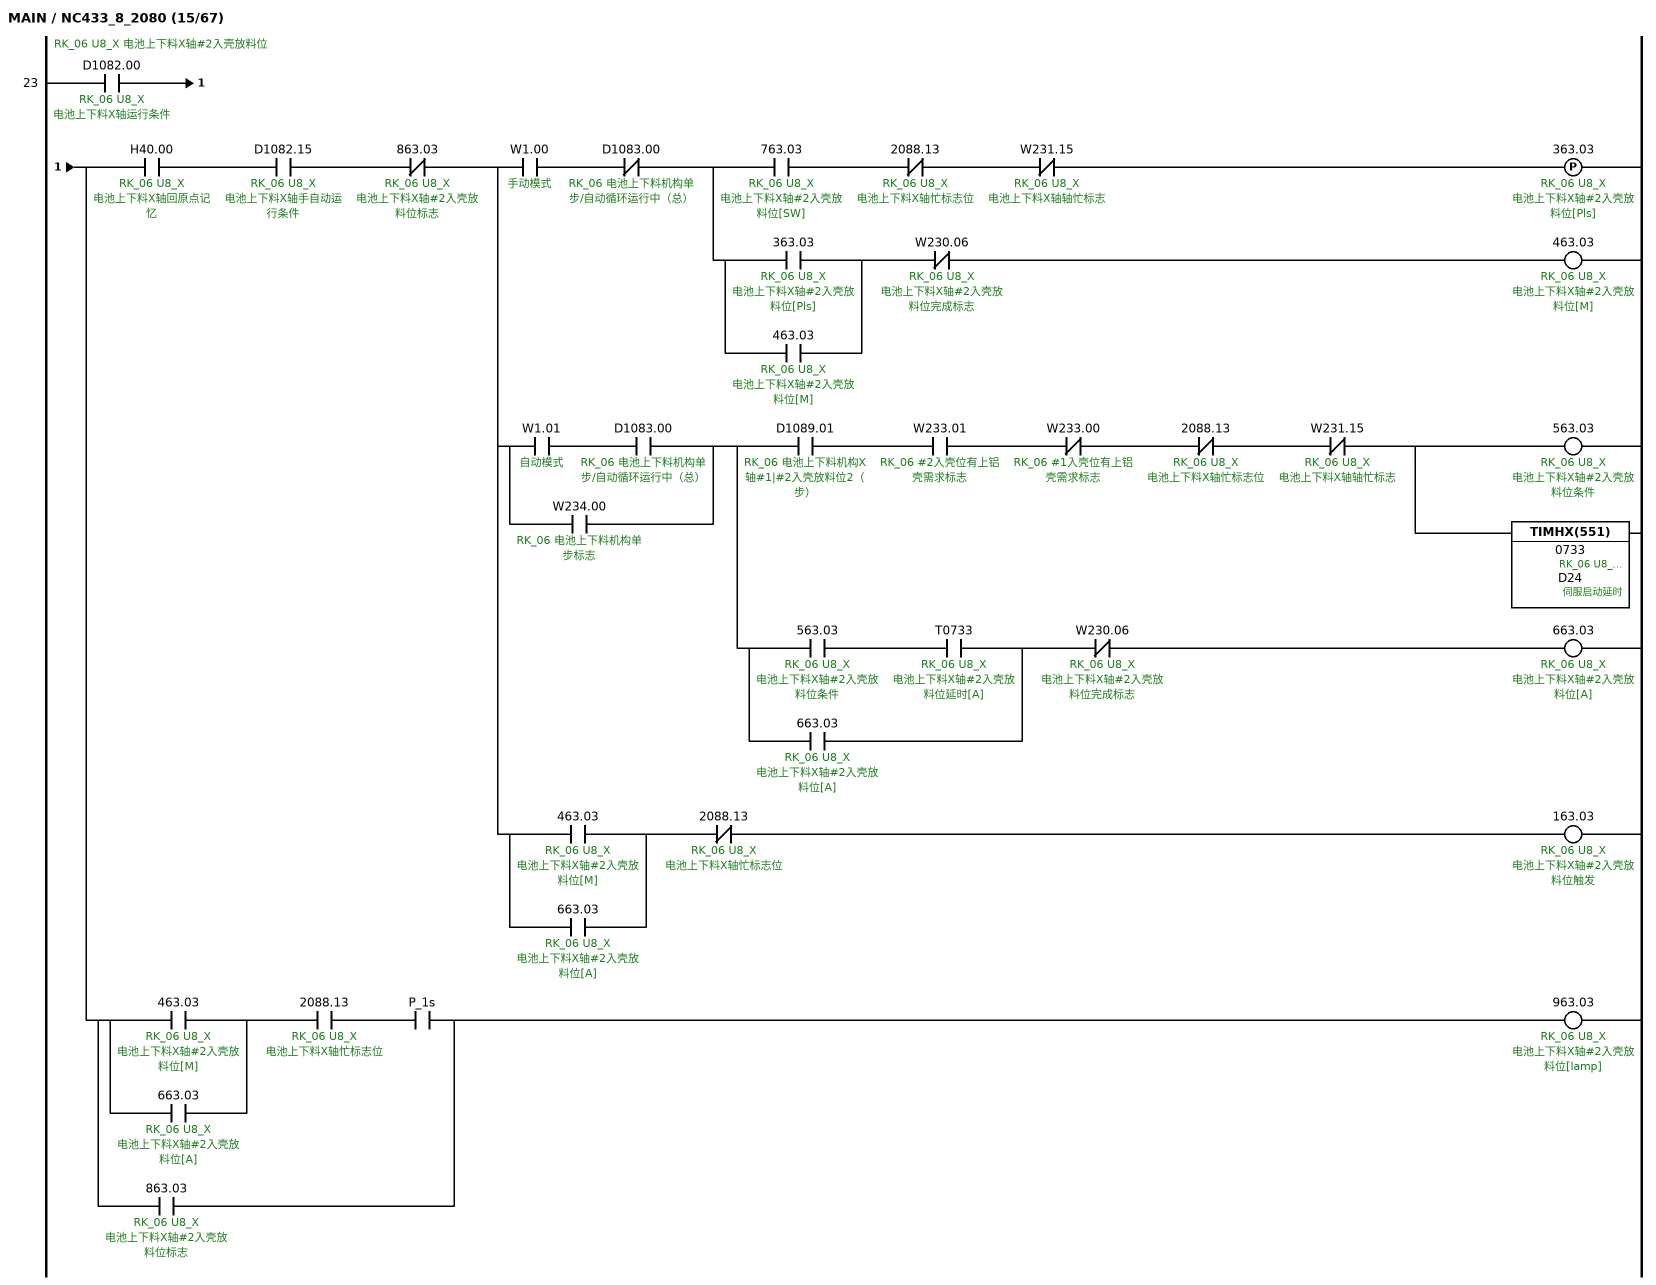
; rung 23: RK_06 U8_X 电池上下料X轴#2入壳放料位
LD D1082.00  ; RK_06 U8_X 电池上下料X轴运行条件
OUT TR0
AND H40.00  ; RK_06 U8_X 电池上下料X轴回原点记忆
AND D1082.15  ; RK_06 U8_X 电池上下料X轴手自动运行条件
ANDNOT 863.03  ; RK_06 U8_X 电池上下料X轴#2入壳放料位标志
OUT TR1
AND W1.00  ; 手动模式
ANDNOT D1083.00  ; RK_06 电池上下料机构单步/自动循环运行中（总）
OUT TR2
AND 763.03  ; RK_06 U8_X 电池上下料X轴#2入壳放料位[SW]
ANDNOT 2088.13  ; RK_06 U8_X 电池上下料X轴忙标志位
ANDNOT W231.15  ; RK_06 U8_X 电池上下料X轴轴忙标志
DIFU(013) 363.03  ; RK_06 U8_X 电池上下料X轴#2入壳放料位[Pls]
LD TR2
LD 363.03  ; RK_06 U8_X 电池上下料X轴#2入壳放料位[Pls]
OR 463.03  ; RK_06 U8_X 电池上下料X轴#2入壳放料位[M]
ANDLD
ANDNOT W230.06  ; RK_06 U8_X 电池上下料X轴#2入壳放料位完成标志
OUT 463.03  ; RK_06 U8_X 电池上下料X轴#2入壳放料位[M]
LD TR1
LD W1.01  ; 自动模式
AND D1083.00  ; RK_06 电池上下料机构单步/自动循环运行中（总）
OR W234.00  ; RK_06 电池上下料机构单步标志
ANDLD
OUT TR2
AND D1089.01  ; RK_06 电池上下料机构X轴#1|#2入壳放料位2（步）
AND W233.01  ; RK_06 #2入壳位有上铝壳需求标志
ANDNOT W233.00  ; RK_06 #1入壳位有上铝壳需求标志
ANDNOT 2088.13  ; RK_06 U8_X 电池上下料X轴忙标志位
ANDNOT W231.15  ; RK_06 U8_X 电池上下料X轴轴忙标志
OUT 563.03  ; RK_06 U8_X 电池上下料X轴#2入壳放料位条件
TIMHX(551) 0733 D24  ; 伺服启动延时, RK_06 U8_X 电池上下料X轴#2入壳放料位延时[A]
LD TR2
LD 563.03  ; RK_06 U8_X 电池上下料X轴#2入壳放料位条件
AND T0733  ; RK_06 U8_X 电池上下料X轴#2入壳放料位延时[A]
OR 663.03  ; RK_06 U8_X 电池上下料X轴#2入壳放料位[A]
ANDLD
ANDNOT W230.06  ; RK_06 U8_X 电池上下料X轴#2入壳放料位完成标志
OUT 663.03  ; RK_06 U8_X 电池上下料X轴#2入壳放料位[A]
LD TR1
LD 463.03  ; RK_06 U8_X 电池上下料X轴#2入壳放料位[M]
OR 663.03  ; RK_06 U8_X 电池上下料X轴#2入壳放料位[A]
ANDLD
ANDNOT 2088.13  ; RK_06 U8_X 电池上下料X轴忙标志位
OUT 163.03  ; RK_06 U8_X 电池上下料X轴#2入壳放料位触发
LD TR0
LD 463.03  ; RK_06 U8_X 电池上下料X轴#2入壳放料位[M]
OR 663.03  ; RK_06 U8_X 电池上下料X轴#2入壳放料位[A]
AND 2088.13  ; RK_06 U8_X 电池上下料X轴忙标志位
AND P_1s
OR 863.03  ; RK_06 U8_X 电池上下料X轴#2入壳放料位标志
ANDLD
OUT 963.03  ; RK_06 U8_X 电池上下料X轴#2入壳放料位[lamp]

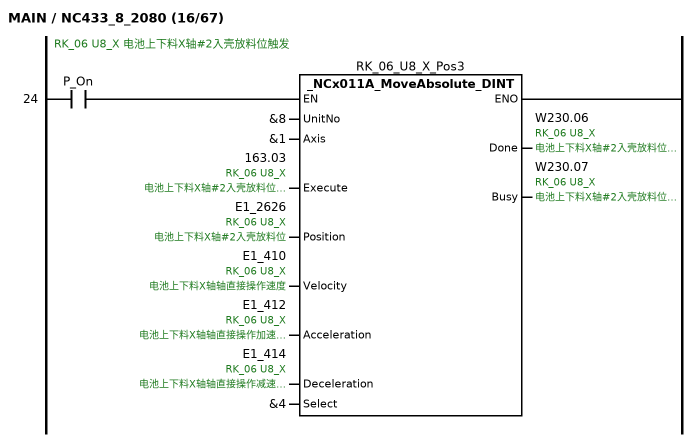
; rung 24: RK_06 U8_X 电池上下料X轴#2入壳放料位触发
LD P_On
CALL RK_06_U8_X_Pos3 : _NCx011A_MoveAbsolute_DINT (UnitNo := &8, Axis := &1, Execute := 163.03, Position := E1_2626, Velocity := E1_410, Acceleration := E1_412, Deceleration := E1_414, Select := &4, Done => W230.06, Busy => W230.07)  ; RK_06 U8_X 电池上下料X轴#2入壳放料位触发, RK_06 U8_X 电池上下料X轴#2入壳放料位, RK_06 U8_X 电池上下料X轴轴直接操作速度, RK_06 U8_X 电池上下料X轴轴直接操作加速时间, RK_06 U8_X 电池上下料X轴轴直接操作减速时间, RK_06 U8_X 电池上下料X轴#2入壳放料位完成标志, RK_06 U8_X 电池上下料X轴#2入壳放料位忙标志

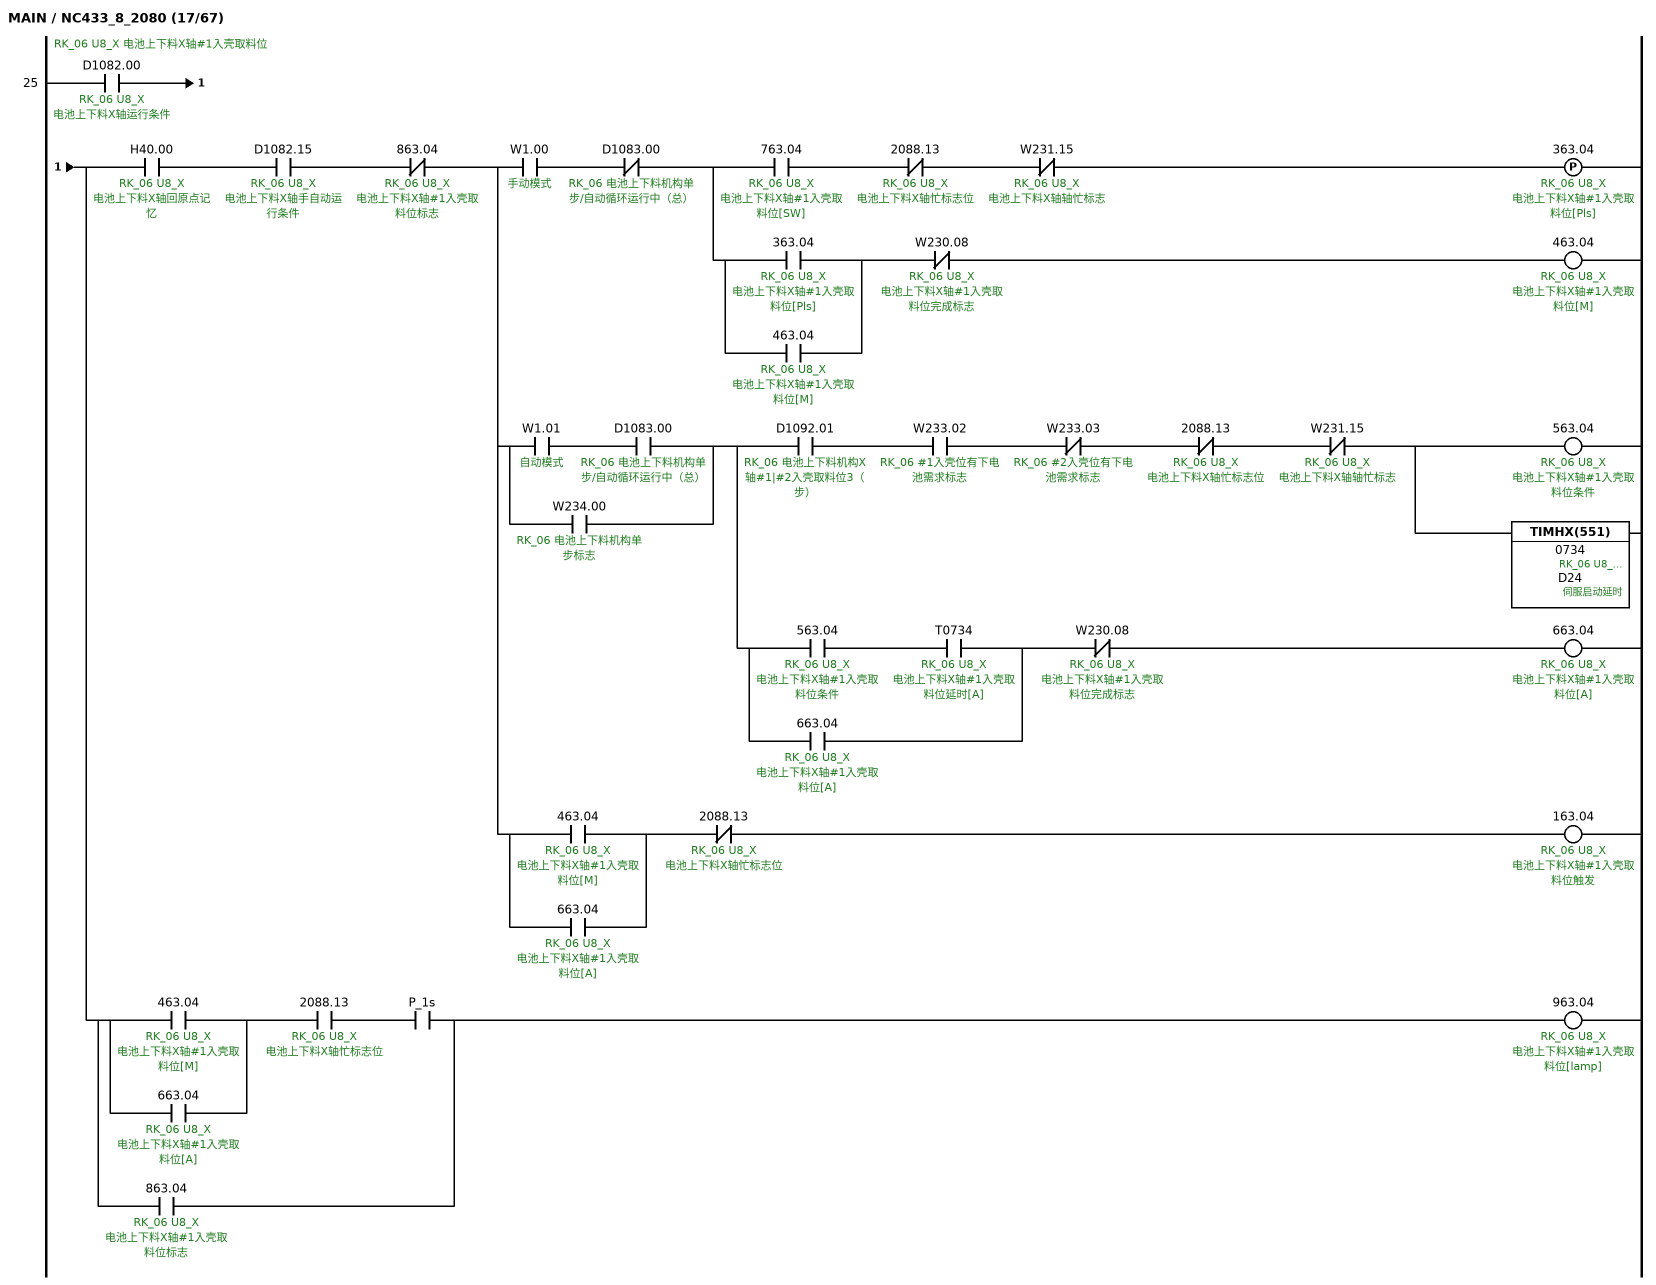
; rung 25: RK_06 U8_X 电池上下料X轴#1入壳取料位
LD D1082.00  ; RK_06 U8_X 电池上下料X轴运行条件
OUT TR0
AND H40.00  ; RK_06 U8_X 电池上下料X轴回原点记忆
AND D1082.15  ; RK_06 U8_X 电池上下料X轴手自动运行条件
ANDNOT 863.04  ; RK_06 U8_X 电池上下料X轴#1入壳取料位标志
OUT TR1
AND W1.00  ; 手动模式
ANDNOT D1083.00  ; RK_06 电池上下料机构单步/自动循环运行中（总）
OUT TR2
AND 763.04  ; RK_06 U8_X 电池上下料X轴#1入壳取料位[SW]
ANDNOT 2088.13  ; RK_06 U8_X 电池上下料X轴忙标志位
ANDNOT W231.15  ; RK_06 U8_X 电池上下料X轴轴忙标志
DIFU(013) 363.04  ; RK_06 U8_X 电池上下料X轴#1入壳取料位[Pls]
LD TR2
LD 363.04  ; RK_06 U8_X 电池上下料X轴#1入壳取料位[Pls]
OR 463.04  ; RK_06 U8_X 电池上下料X轴#1入壳取料位[M]
ANDLD
ANDNOT W230.08  ; RK_06 U8_X 电池上下料X轴#1入壳取料位完成标志
OUT 463.04  ; RK_06 U8_X 电池上下料X轴#1入壳取料位[M]
LD TR1
LD W1.01  ; 自动模式
AND D1083.00  ; RK_06 电池上下料机构单步/自动循环运行中（总）
OR W234.00  ; RK_06 电池上下料机构单步标志
ANDLD
OUT TR2
AND D1092.01  ; RK_06 电池上下料机构X轴#1|#2入壳取料位3（步）
AND W233.02  ; RK_06 #1入壳位有下电池需求标志
ANDNOT W233.03  ; RK_06 #2入壳位有下电池需求标志
ANDNOT 2088.13  ; RK_06 U8_X 电池上下料X轴忙标志位
ANDNOT W231.15  ; RK_06 U8_X 电池上下料X轴轴忙标志
OUT 563.04  ; RK_06 U8_X 电池上下料X轴#1入壳取料位条件
TIMHX(551) 0734 D24  ; 伺服启动延时, RK_06 U8_X 电池上下料X轴#1入壳取料位延时[A]
LD TR2
LD 563.04  ; RK_06 U8_X 电池上下料X轴#1入壳取料位条件
AND T0734  ; RK_06 U8_X 电池上下料X轴#1入壳取料位延时[A]
OR 663.04  ; RK_06 U8_X 电池上下料X轴#1入壳取料位[A]
ANDLD
ANDNOT W230.08  ; RK_06 U8_X 电池上下料X轴#1入壳取料位完成标志
OUT 663.04  ; RK_06 U8_X 电池上下料X轴#1入壳取料位[A]
LD TR1
LD 463.04  ; RK_06 U8_X 电池上下料X轴#1入壳取料位[M]
OR 663.04  ; RK_06 U8_X 电池上下料X轴#1入壳取料位[A]
ANDLD
ANDNOT 2088.13  ; RK_06 U8_X 电池上下料X轴忙标志位
OUT 163.04  ; RK_06 U8_X 电池上下料X轴#1入壳取料位触发
LD TR0
LD 463.04  ; RK_06 U8_X 电池上下料X轴#1入壳取料位[M]
OR 663.04  ; RK_06 U8_X 电池上下料X轴#1入壳取料位[A]
AND 2088.13  ; RK_06 U8_X 电池上下料X轴忙标志位
AND P_1s
OR 863.04  ; RK_06 U8_X 电池上下料X轴#1入壳取料位标志
ANDLD
OUT 963.04  ; RK_06 U8_X 电池上下料X轴#1入壳取料位[lamp]

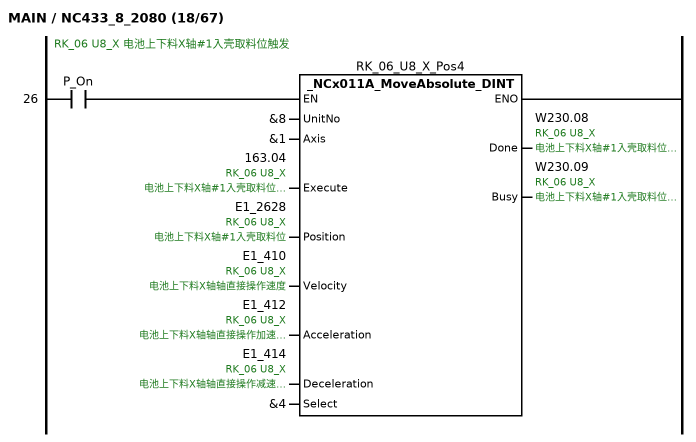
; rung 26: RK_06 U8_X 电池上下料X轴#1入壳取料位触发
LD P_On
CALL RK_06_U8_X_Pos4 : _NCx011A_MoveAbsolute_DINT (UnitNo := &8, Axis := &1, Execute := 163.04, Position := E1_2628, Velocity := E1_410, Acceleration := E1_412, Deceleration := E1_414, Select := &4, Done => W230.08, Busy => W230.09)  ; RK_06 U8_X 电池上下料X轴#1入壳取料位触发, RK_06 U8_X 电池上下料X轴#1入壳取料位, RK_06 U8_X 电池上下料X轴轴直接操作速度, RK_06 U8_X 电池上下料X轴轴直接操作加速时间, RK_06 U8_X 电池上下料X轴轴直接操作减速时间, RK_06 U8_X 电池上下料X轴#1入壳取料位完成标志, RK_06 U8_X 电池上下料X轴#1入壳取料位忙标志

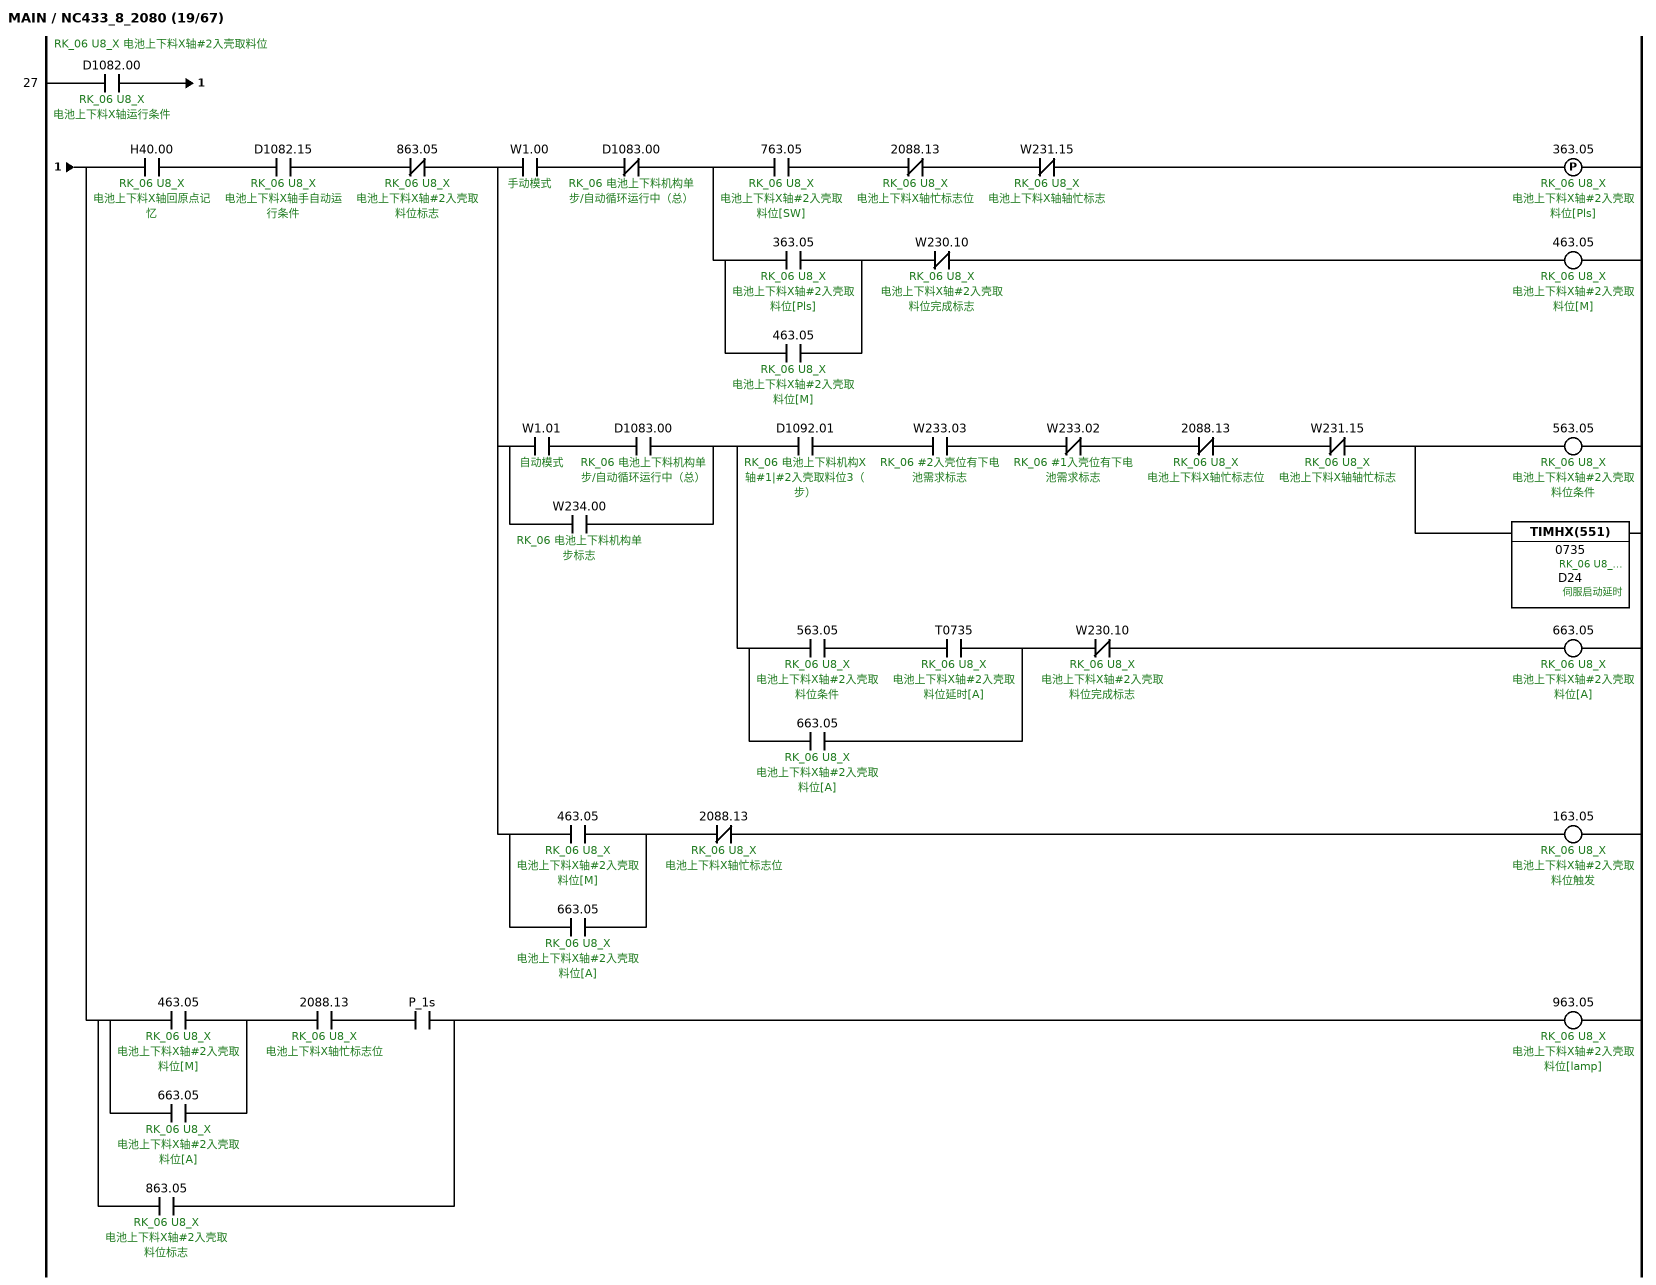
; rung 27: RK_06 U8_X 电池上下料X轴#2入壳取料位
LD D1082.00  ; RK_06 U8_X 电池上下料X轴运行条件
OUT TR0
AND H40.00  ; RK_06 U8_X 电池上下料X轴回原点记忆
AND D1082.15  ; RK_06 U8_X 电池上下料X轴手自动运行条件
ANDNOT 863.05  ; RK_06 U8_X 电池上下料X轴#2入壳取料位标志
OUT TR1
AND W1.00  ; 手动模式
ANDNOT D1083.00  ; RK_06 电池上下料机构单步/自动循环运行中（总）
OUT TR2
AND 763.05  ; RK_06 U8_X 电池上下料X轴#2入壳取料位[SW]
ANDNOT 2088.13  ; RK_06 U8_X 电池上下料X轴忙标志位
ANDNOT W231.15  ; RK_06 U8_X 电池上下料X轴轴忙标志
DIFU(013) 363.05  ; RK_06 U8_X 电池上下料X轴#2入壳取料位[Pls]
LD TR2
LD 363.05  ; RK_06 U8_X 电池上下料X轴#2入壳取料位[Pls]
OR 463.05  ; RK_06 U8_X 电池上下料X轴#2入壳取料位[M]
ANDLD
ANDNOT W230.10  ; RK_06 U8_X 电池上下料X轴#2入壳取料位完成标志
OUT 463.05  ; RK_06 U8_X 电池上下料X轴#2入壳取料位[M]
LD TR1
LD W1.01  ; 自动模式
AND D1083.00  ; RK_06 电池上下料机构单步/自动循环运行中（总）
OR W234.00  ; RK_06 电池上下料机构单步标志
ANDLD
OUT TR2
AND D1092.01  ; RK_06 电池上下料机构X轴#1|#2入壳取料位3（步）
AND W233.03  ; RK_06 #2入壳位有下电池需求标志
ANDNOT W233.02  ; RK_06 #1入壳位有下电池需求标志
ANDNOT 2088.13  ; RK_06 U8_X 电池上下料X轴忙标志位
ANDNOT W231.15  ; RK_06 U8_X 电池上下料X轴轴忙标志
OUT 563.05  ; RK_06 U8_X 电池上下料X轴#2入壳取料位条件
TIMHX(551) 0735 D24  ; 伺服启动延时, RK_06 U8_X 电池上下料X轴#2入壳取料位延时[A]
LD TR2
LD 563.05  ; RK_06 U8_X 电池上下料X轴#2入壳取料位条件
AND T0735  ; RK_06 U8_X 电池上下料X轴#2入壳取料位延时[A]
OR 663.05  ; RK_06 U8_X 电池上下料X轴#2入壳取料位[A]
ANDLD
ANDNOT W230.10  ; RK_06 U8_X 电池上下料X轴#2入壳取料位完成标志
OUT 663.05  ; RK_06 U8_X 电池上下料X轴#2入壳取料位[A]
LD TR1
LD 463.05  ; RK_06 U8_X 电池上下料X轴#2入壳取料位[M]
OR 663.05  ; RK_06 U8_X 电池上下料X轴#2入壳取料位[A]
ANDLD
ANDNOT 2088.13  ; RK_06 U8_X 电池上下料X轴忙标志位
OUT 163.05  ; RK_06 U8_X 电池上下料X轴#2入壳取料位触发
LD TR0
LD 463.05  ; RK_06 U8_X 电池上下料X轴#2入壳取料位[M]
OR 663.05  ; RK_06 U8_X 电池上下料X轴#2入壳取料位[A]
AND 2088.13  ; RK_06 U8_X 电池上下料X轴忙标志位
AND P_1s
OR 863.05  ; RK_06 U8_X 电池上下料X轴#2入壳取料位标志
ANDLD
OUT 963.05  ; RK_06 U8_X 电池上下料X轴#2入壳取料位[lamp]

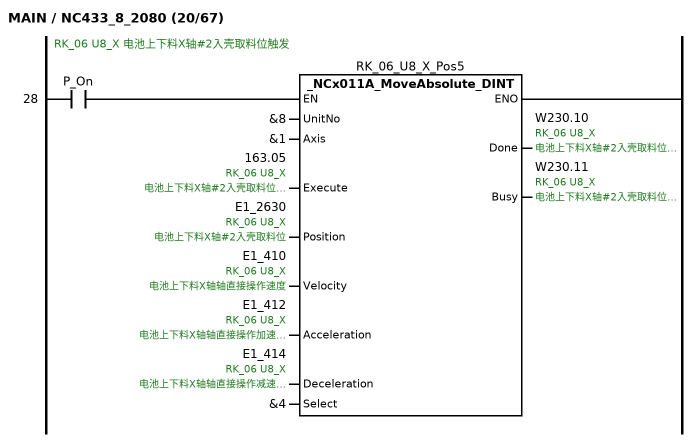
; rung 28: RK_06 U8_X 电池上下料X轴#2入壳取料位触发
LD P_On
CALL RK_06_U8_X_Pos5 : _NCx011A_MoveAbsolute_DINT (UnitNo := &8, Axis := &1, Execute := 163.05, Position := E1_2630, Velocity := E1_410, Acceleration := E1_412, Deceleration := E1_414, Select := &4, Done => W230.10, Busy => W230.11)  ; RK_06 U8_X 电池上下料X轴#2入壳取料位触发, RK_06 U8_X 电池上下料X轴#2入壳取料位, RK_06 U8_X 电池上下料X轴轴直接操作速度, RK_06 U8_X 电池上下料X轴轴直接操作加速时间, RK_06 U8_X 电池上下料X轴轴直接操作减速时间, RK_06 U8_X 电池上下料X轴#2入壳取料位完成标志, RK_06 U8_X 电池上下料X轴#2入壳取料位忙标志

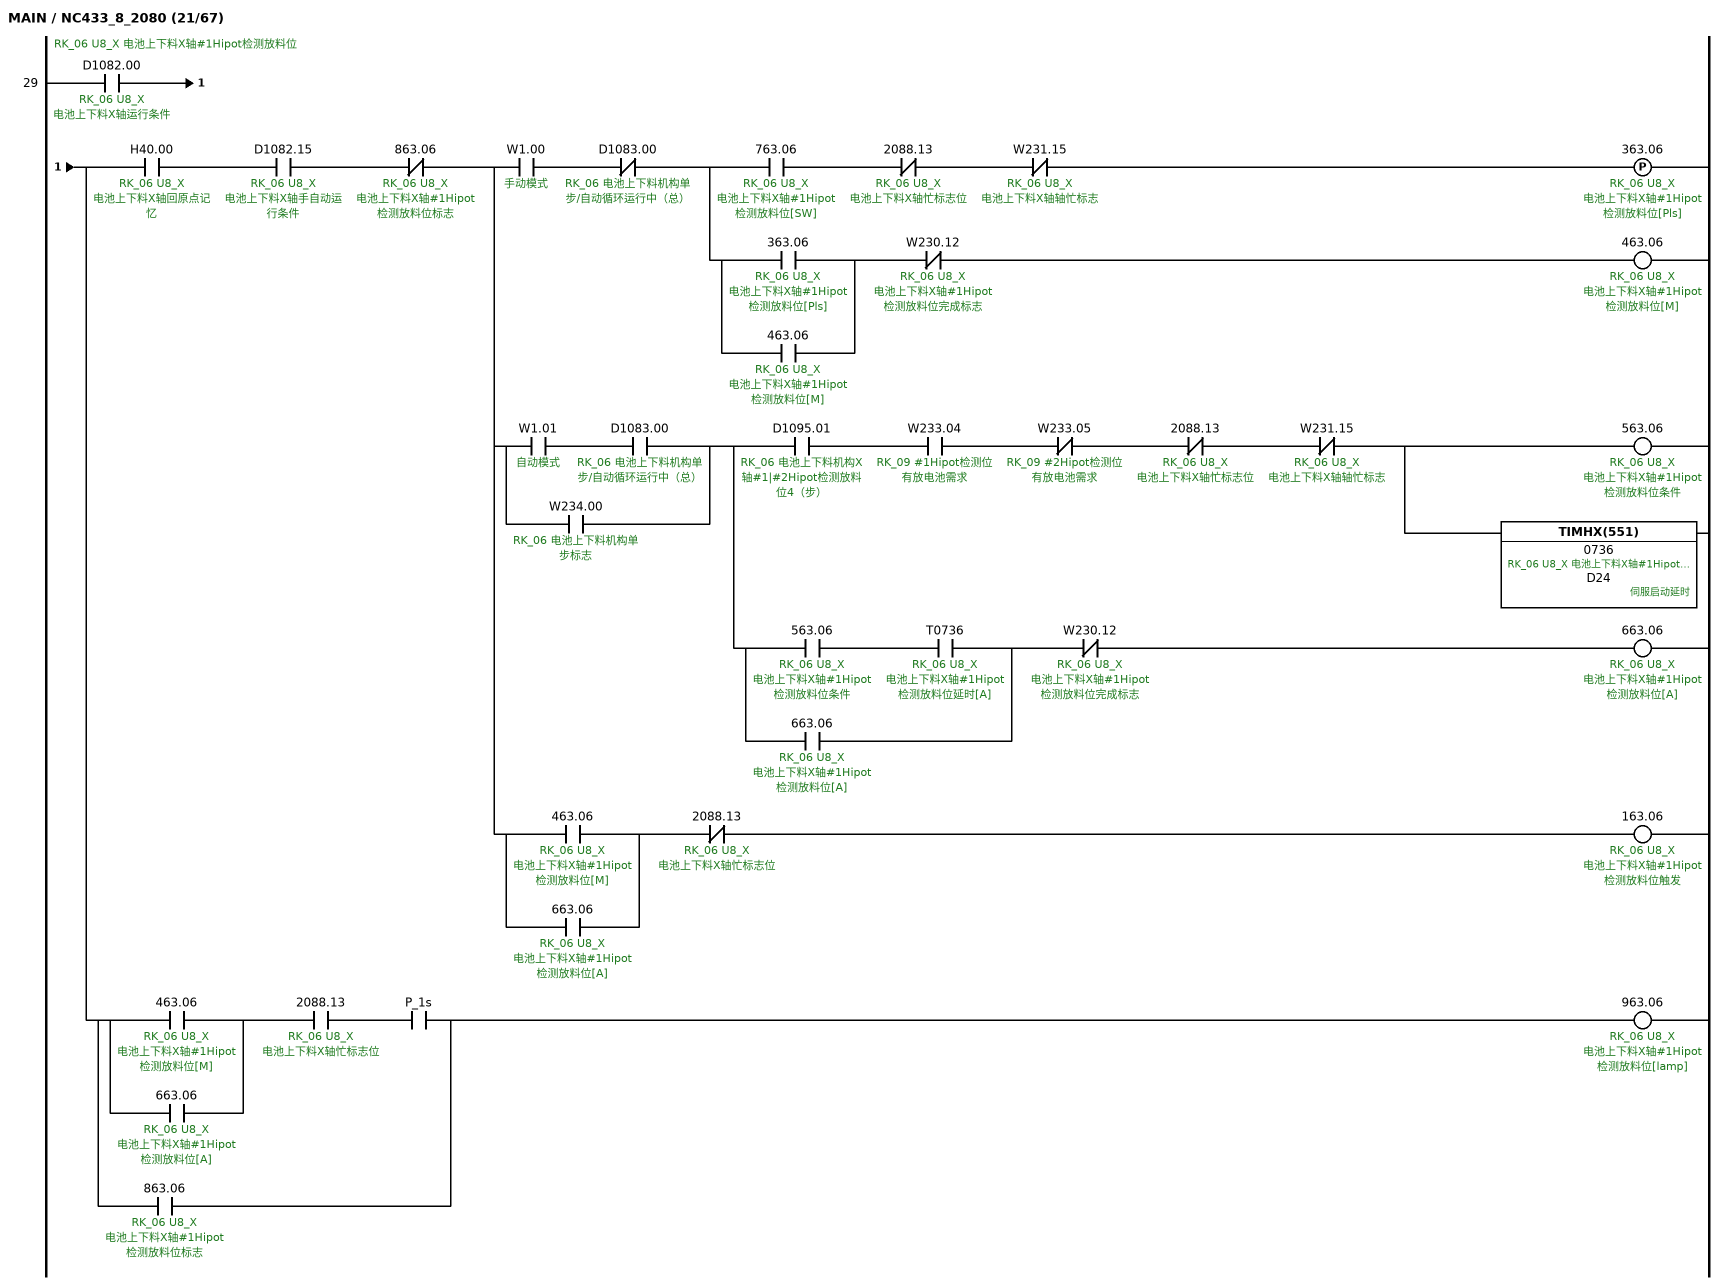
; rung 29: RK_06 U8_X 电池上下料X轴#1Hipot检测放料位
LD D1082.00  ; RK_06 U8_X 电池上下料X轴运行条件
OUT TR0
AND H40.00  ; RK_06 U8_X 电池上下料X轴回原点记忆
AND D1082.15  ; RK_06 U8_X 电池上下料X轴手自动运行条件
ANDNOT 863.06  ; RK_06 U8_X 电池上下料X轴#1Hipot检测放料位标志
OUT TR1
AND W1.00  ; 手动模式
ANDNOT D1083.00  ; RK_06 电池上下料机构单步/自动循环运行中（总）
OUT TR2
AND 763.06  ; RK_06 U8_X 电池上下料X轴#1Hipot检测放料位[SW]
ANDNOT 2088.13  ; RK_06 U8_X 电池上下料X轴忙标志位
ANDNOT W231.15  ; RK_06 U8_X 电池上下料X轴轴忙标志
DIFU(013) 363.06  ; RK_06 U8_X 电池上下料X轴#1Hipot检测放料位[Pls]
LD TR2
LD 363.06  ; RK_06 U8_X 电池上下料X轴#1Hipot检测放料位[Pls]
OR 463.06  ; RK_06 U8_X 电池上下料X轴#1Hipot检测放料位[M]
ANDLD
ANDNOT W230.12  ; RK_06 U8_X 电池上下料X轴#1Hipot检测放料位完成标志
OUT 463.06  ; RK_06 U8_X 电池上下料X轴#1Hipot检测放料位[M]
LD TR1
LD W1.01  ; 自动模式
AND D1083.00  ; RK_06 电池上下料机构单步/自动循环运行中（总）
OR W234.00  ; RK_06 电池上下料机构单步标志
ANDLD
OUT TR2
AND D1095.01  ; RK_06 电池上下料机构X轴#1|#2Hipot检测放料位4（步）
AND W233.04  ; RK_09 #1Hipot检测位有放电池需求
ANDNOT W233.05  ; RK_09 #2Hipot检测位有放电池需求
ANDNOT 2088.13  ; RK_06 U8_X 电池上下料X轴忙标志位
ANDNOT W231.15  ; RK_06 U8_X 电池上下料X轴轴忙标志
OUT 563.06  ; RK_06 U8_X 电池上下料X轴#1Hipot检测放料位条件
TIMHX(551) 0736 D24  ; 伺服启动延时, RK_06 U8_X 电池上下料X轴#1Hipot检测放料位延时[A]
LD TR2
LD 563.06  ; RK_06 U8_X 电池上下料X轴#1Hipot检测放料位条件
AND T0736  ; RK_06 U8_X 电池上下料X轴#1Hipot检测放料位延时[A]
OR 663.06  ; RK_06 U8_X 电池上下料X轴#1Hipot检测放料位[A]
ANDLD
ANDNOT W230.12  ; RK_06 U8_X 电池上下料X轴#1Hipot检测放料位完成标志
OUT 663.06  ; RK_06 U8_X 电池上下料X轴#1Hipot检测放料位[A]
LD TR1
LD 463.06  ; RK_06 U8_X 电池上下料X轴#1Hipot检测放料位[M]
OR 663.06  ; RK_06 U8_X 电池上下料X轴#1Hipot检测放料位[A]
ANDLD
ANDNOT 2088.13  ; RK_06 U8_X 电池上下料X轴忙标志位
OUT 163.06  ; RK_06 U8_X 电池上下料X轴#1Hipot检测放料位触发
LD TR0
LD 463.06  ; RK_06 U8_X 电池上下料X轴#1Hipot检测放料位[M]
OR 663.06  ; RK_06 U8_X 电池上下料X轴#1Hipot检测放料位[A]
AND 2088.13  ; RK_06 U8_X 电池上下料X轴忙标志位
AND P_1s
OR 863.06  ; RK_06 U8_X 电池上下料X轴#1Hipot检测放料位标志
ANDLD
OUT 963.06  ; RK_06 U8_X 电池上下料X轴#1Hipot检测放料位[lamp]

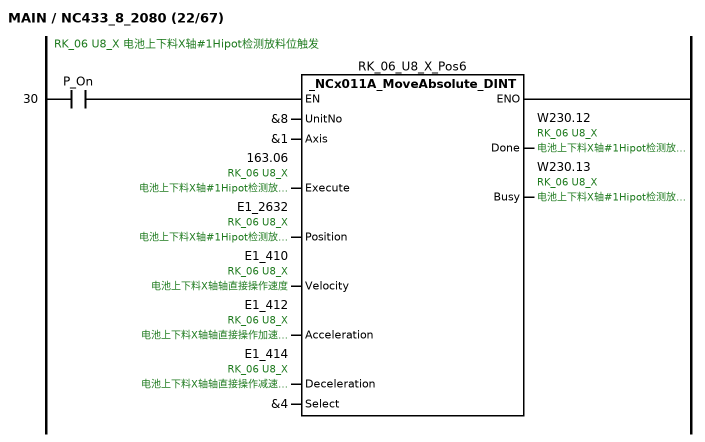
; rung 30: RK_06 U8_X 电池上下料X轴#1Hipot检测放料位触发
LD P_On
CALL RK_06_U8_X_Pos6 : _NCx011A_MoveAbsolute_DINT (UnitNo := &8, Axis := &1, Execute := 163.06, Position := E1_2632, Velocity := E1_410, Acceleration := E1_412, Deceleration := E1_414, Select := &4, Done => W230.12, Busy => W230.13)  ; RK_06 U8_X 电池上下料X轴#1Hipot检测放料位触发, RK_06 U8_X 电池上下料X轴#1Hipot检测放料位, RK_06 U8_X 电池上下料X轴轴直接操作速度, RK_06 U8_X 电池上下料X轴轴直接操作加速时间, RK_06 U8_X 电池上下料X轴轴直接操作减速时间, RK_06 U8_X 电池上下料X轴#1Hipot检测放料位完成标志, RK_06 U8_X 电池上下料X轴#1Hipot检测放料位忙标志

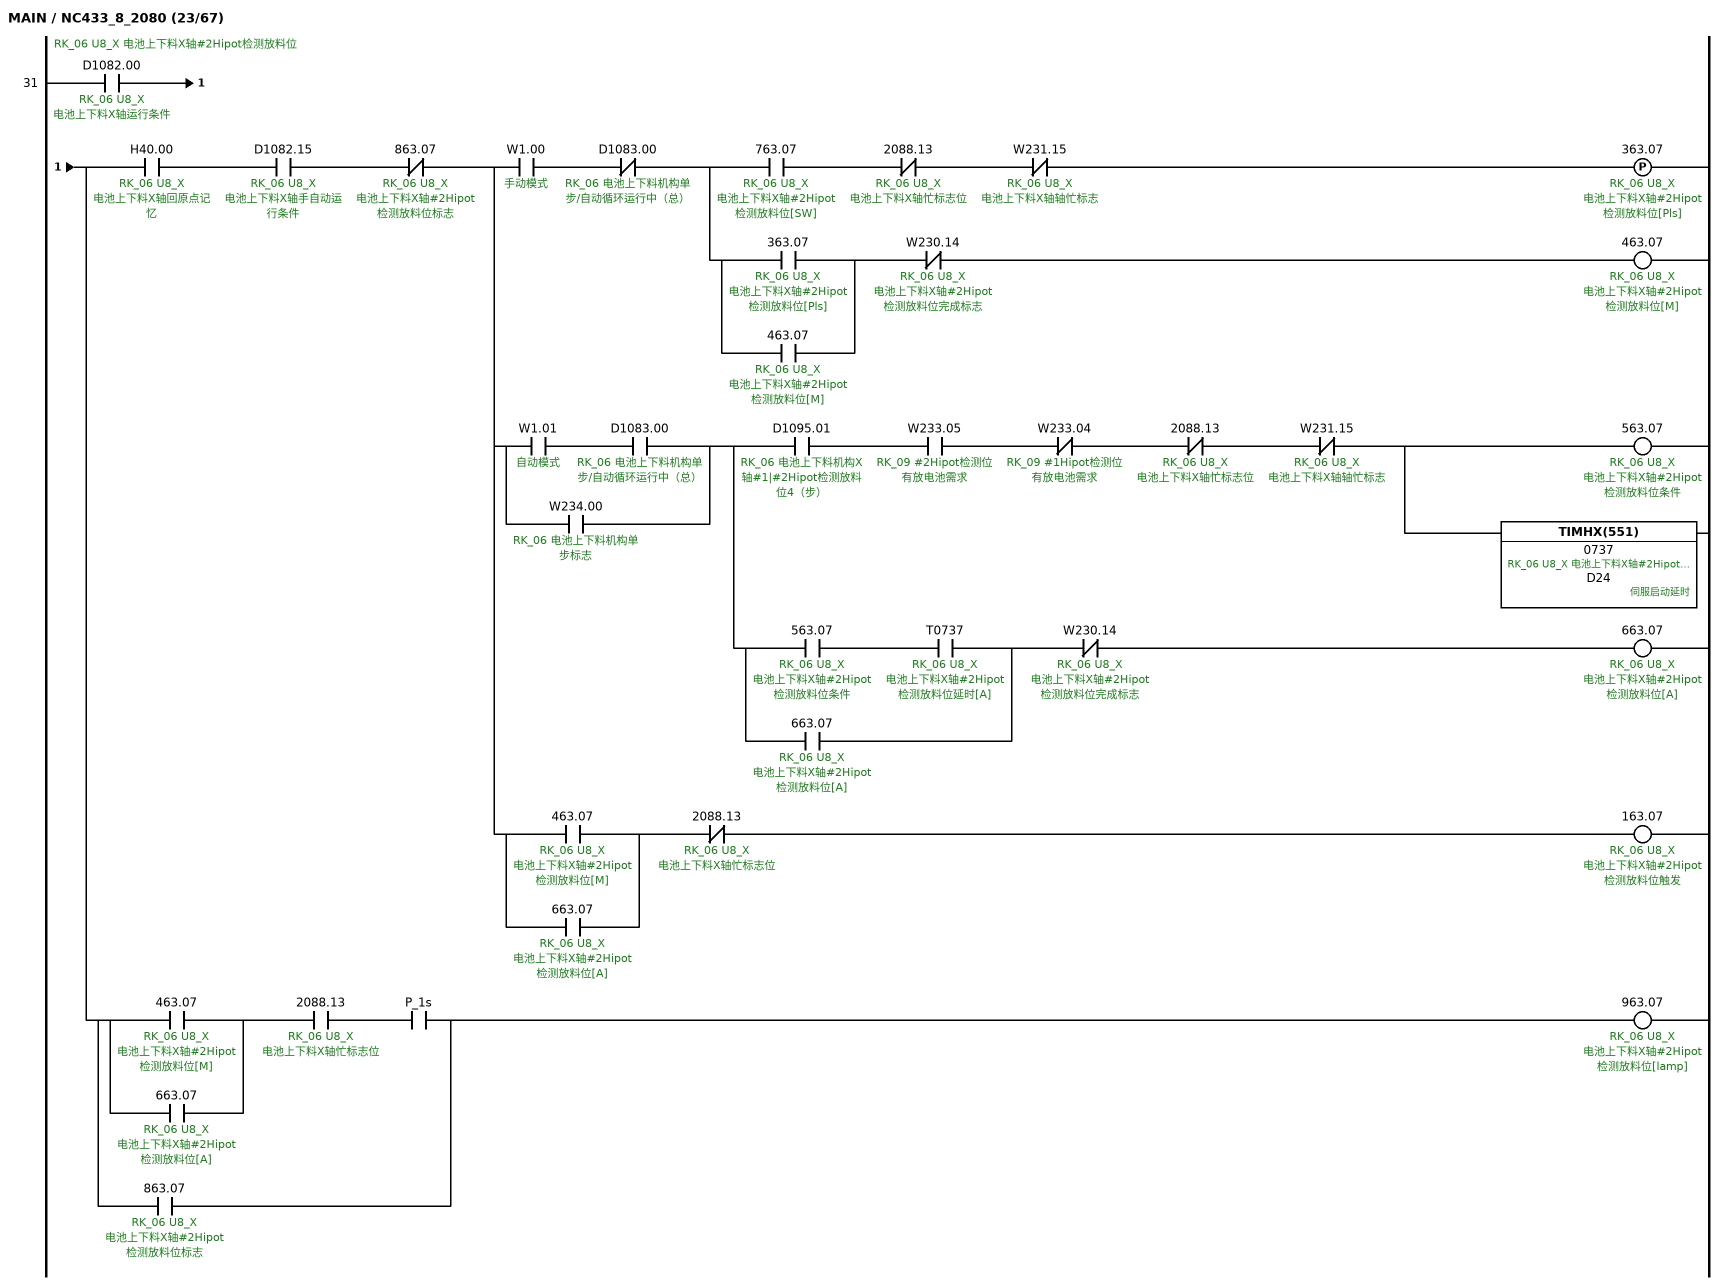
; rung 31: RK_06 U8_X 电池上下料X轴#2Hipot检测放料位
LD D1082.00  ; RK_06 U8_X 电池上下料X轴运行条件
OUT TR0
AND H40.00  ; RK_06 U8_X 电池上下料X轴回原点记忆
AND D1082.15  ; RK_06 U8_X 电池上下料X轴手自动运行条件
ANDNOT 863.07  ; RK_06 U8_X 电池上下料X轴#2Hipot检测放料位标志
OUT TR1
AND W1.00  ; 手动模式
ANDNOT D1083.00  ; RK_06 电池上下料机构单步/自动循环运行中（总）
OUT TR2
AND 763.07  ; RK_06 U8_X 电池上下料X轴#2Hipot检测放料位[SW]
ANDNOT 2088.13  ; RK_06 U8_X 电池上下料X轴忙标志位
ANDNOT W231.15  ; RK_06 U8_X 电池上下料X轴轴忙标志
DIFU(013) 363.07  ; RK_06 U8_X 电池上下料X轴#2Hipot检测放料位[Pls]
LD TR2
LD 363.07  ; RK_06 U8_X 电池上下料X轴#2Hipot检测放料位[Pls]
OR 463.07  ; RK_06 U8_X 电池上下料X轴#2Hipot检测放料位[M]
ANDLD
ANDNOT W230.14  ; RK_06 U8_X 电池上下料X轴#2Hipot检测放料位完成标志
OUT 463.07  ; RK_06 U8_X 电池上下料X轴#2Hipot检测放料位[M]
LD TR1
LD W1.01  ; 自动模式
AND D1083.00  ; RK_06 电池上下料机构单步/自动循环运行中（总）
OR W234.00  ; RK_06 电池上下料机构单步标志
ANDLD
OUT TR2
AND D1095.01  ; RK_06 电池上下料机构X轴#1|#2Hipot检测放料位4（步）
AND W233.05  ; RK_09 #2Hipot检测位有放电池需求
ANDNOT W233.04  ; RK_09 #1Hipot检测位有放电池需求
ANDNOT 2088.13  ; RK_06 U8_X 电池上下料X轴忙标志位
ANDNOT W231.15  ; RK_06 U8_X 电池上下料X轴轴忙标志
OUT 563.07  ; RK_06 U8_X 电池上下料X轴#2Hipot检测放料位条件
TIMHX(551) 0737 D24  ; 伺服启动延时, RK_06 U8_X 电池上下料X轴#2Hipot检测放料位延时[A]
LD TR2
LD 563.07  ; RK_06 U8_X 电池上下料X轴#2Hipot检测放料位条件
AND T0737  ; RK_06 U8_X 电池上下料X轴#2Hipot检测放料位延时[A]
OR 663.07  ; RK_06 U8_X 电池上下料X轴#2Hipot检测放料位[A]
ANDLD
ANDNOT W230.14  ; RK_06 U8_X 电池上下料X轴#2Hipot检测放料位完成标志
OUT 663.07  ; RK_06 U8_X 电池上下料X轴#2Hipot检测放料位[A]
LD TR1
LD 463.07  ; RK_06 U8_X 电池上下料X轴#2Hipot检测放料位[M]
OR 663.07  ; RK_06 U8_X 电池上下料X轴#2Hipot检测放料位[A]
ANDLD
ANDNOT 2088.13  ; RK_06 U8_X 电池上下料X轴忙标志位
OUT 163.07  ; RK_06 U8_X 电池上下料X轴#2Hipot检测放料位触发
LD TR0
LD 463.07  ; RK_06 U8_X 电池上下料X轴#2Hipot检测放料位[M]
OR 663.07  ; RK_06 U8_X 电池上下料X轴#2Hipot检测放料位[A]
AND 2088.13  ; RK_06 U8_X 电池上下料X轴忙标志位
AND P_1s
OR 863.07  ; RK_06 U8_X 电池上下料X轴#2Hipot检测放料位标志
ANDLD
OUT 963.07  ; RK_06 U8_X 电池上下料X轴#2Hipot检测放料位[lamp]

